LIN{ E6POS: X 728.6422, Y 47.5546, Z -92.0150, A 0, B 90, C 0, E1 0, E2 0, E3 0, E4 0 } C_DIS
LIN{ E6POS: X 729.6150, Y 47.3233, Z -92.0150, A 0, B 90, C 0, E1 0, E2 0, E3 0, E4 0 } C_DIS
LIN{ E6POS: X 730.5879, Y 47.0919, Z -92.0150, A 0, B 90, C 0, E1 0, E2 0, E3 0, E4 0 } C_DIS
LIN{ E6POS: X 731.5608, Y 46.8606, Z -92.0150, A 0, B 90, C 0, E1 0, E2 0, E3 0, E4 0 } C_DIS
LIN{ E6POS: X 731.5744, Y 46.8574, Z -92.0150, A 0, B 90, C 0, E1 0, E2 0, E3 0, E4 0 } C_DIS
LIN{ E6POS: X 732.5446, Y 46.6148, Z -92.0150, A 0, B 90, C 0, E1 0, E2 0, E3 0, E4 0 } C_DIS
LIN{ E6POS: X 733.5147, Y 46.3723, Z -92.0150, A 0, B 90, C 0, E1 0, E2 0, E3 0, E4 0 } C_DIS
LIN{ E6POS: X 734.4849, Y 46.1297, Z -92.0150, A 0, B 90, C 0, E1 0, E2 0, E3 0, E4 0 } C_DIS
LIN{ E6POS: X 735.4550, Y 45.8872, Z -92.0150, A 0, B 90, C 0, E1 0, E2 0, E3 0, E4 0 } C_DIS
LIN{ E6POS: X 736.4251, Y 45.6447, Z -92.0150, A 0, B 90, C 0, E1 0, E2 0, E3 0, E4 0 } C_DIS
LIN{ E6POS: X 737.3953, Y 45.4021, Z -92.0150, A 0, B 90, C 0, E1 0, E2 0, E3 0, E4 0 } C_DIS
LIN{ E6POS: X 738.3654, Y 45.1596, Z -92.0150, A 0, B 90, C 0, E1 0, E2 0, E3 0, E4 0 } C_DIS
LIN{ E6POS: X 739.3356, Y 44.9170, Z -92.0150, A 0, B 90, C 0, E1 0, E2 0, E3 0, E4 0 } C_DIS
LIN{ E6POS: X 740.3057, Y 44.6745, Z -92.0150, A 0, B 90, C 0, E1 0, E2 0, E3 0, E4 0 } C_DIS
LIN{ E6POS: X 740.8582, Y 44.5364, Z -92.0150, A 0, B 90, C 0, E1 0, E2 0, E3 0, E4 0 } C_DIS
LIN{ E6POS: X 741.8351, Y 44.3226, Z -92.0150, A 0, B 90, C 0, E1 0, E2 0, E3 0, E4 0 } C_DIS
LIN{ E6POS: X 742.8120, Y 44.1088, Z -92.0150, A 0, B 90, C 0, E1 0, E2 0, E3 0, E4 0 } C_DIS
LIN{ E6POS: X 743.7889, Y 43.8950, Z -92.0150, A 0, B 90, C 0, E1 0, E2 0, E3 0, E4 0 } C_DIS
LIN{ E6POS: X 744.7658, Y 43.6813, Z -92.0150, A 0, B 90, C 0, E1 0, E2 0, E3 0, E4 0 } C_DIS
LIN{ E6POS: X 744.9749, Y 43.6355, Z -92.0150, A 0, B 90, C 0, E1 0, E2 0, E3 0, E4 0 } C_DIS
LIN{ E6POS: X 745.9497, Y 43.4121, Z -92.0150, A 0, B 90, C 0, E1 0, E2 0, E3 0, E4 0 } C_DIS
LIN{ E6POS: X 746.9244, Y 43.1888, Z -92.0150, A 0, B 90, C 0, E1 0, E2 0, E3 0, E4 0 } C_DIS
LIN{ E6POS: X 747.8991, Y 42.9654, Z -92.0150, A 0, B 90, C 0, E1 0, E2 0, E3 0, E4 0 } C_DIS
LIN{ E6POS: X 748.8739, Y 42.7421, Z -92.0150, A 0, B 90, C 0, E1 0, E2 0, E3 0, E4 0 } C_DIS
LIN{ E6POS: X 749.8486, Y 42.5187, Z -92.0150, A 0, B 90, C 0, E1 0, E2 0, E3 0, E4 0 } C_DIS
LIN{ E6POS: X 750.8233, Y 42.2954, Z -92.0150, A 0, B 90, C 0, E1 0, E2 0, E3 0, E4 0 } C_DIS
LIN{ E6POS: X 751.7981, Y 42.0720, Z -92.0150, A 0, B 90, C 0, E1 0, E2 0, E3 0, E4 0 } C_DIS
LIN{ E6POS: X 752.7728, Y 41.8487, Z -92.0150, A 0, B 90, C 0, E1 0, E2 0, E3 0, E4 0 } C_DIS
LIN{ E6POS: X 753.7476, Y 41.6253, Z -92.0150, A 0, B 90, C 0, E1 0, E2 0, E3 0, E4 0 } C_DIS
LIN{ E6POS: X 754.7223, Y 41.4020, Z -92.0150, A 0, B 90, C 0, E1 0, E2 0, E3 0, E4 0 } C_DIS
LIN{ E6POS: X 754.8028, Y 41.3835, Z -92.0150, A 0, B 90, C 0, E1 0, E2 0, E3 0, E4 0 } C_DIS
LIN{ E6POS: X 755.7861, Y 41.2018, Z -92.0150, A 0, B 90, C 0, E1 0, E2 0, E3 0, E4 0 } C_DIS
LIN{ E6POS: X 756.7695, Y 41.0200, Z -92.0150, A 0, B 90, C 0, E1 0, E2 0, E3 0, E4 0 } C_DIS
LIN{ E6POS: X 757.7528, Y 40.8382, Z -92.0150, A 0, B 90, C 0, E1 0, E2 0, E3 0, E4 0 } C_DIS
LIN{ E6POS: X 758.6031, Y 40.6810, Z -92.0150, A 0, B 90, C 0, E1 0, E2 0, E3 0, E4 0 } C_DIS
LIN{ E6POS: X 759.5852, Y 40.4926, Z -92.0150, A 0, B 90, C 0, E1 0, E2 0, E3 0, E4 0 } C_DIS
LIN{ E6POS: X 760.5673, Y 40.3042, Z -92.0150, A 0, B 90, C 0, E1 0, E2 0, E3 0, E4 0 } C_DIS
LIN{ E6POS: X 761.5493, Y 40.1158, Z -92.0150, A 0, B 90, C 0, E1 0, E2 0, E3 0, E4 0 } C_DIS
LIN{ E6POS: X 762.5314, Y 39.9273, Z -92.0150, A 0, B 90, C 0, E1 0, E2 0, E3 0, E4 0 } C_DIS
LIN{ E6POS: X 763.5135, Y 39.7389, Z -92.0150, A 0, B 90, C 0, E1 0, E2 0, E3 0, E4 0 } C_DIS
LIN{ E6POS: X 764.4956, Y 39.5505, Z -92.0150, A 0, B 90, C 0, E1 0, E2 0, E3 0, E4 0 } C_DIS
LIN{ E6POS: X 765.4777, Y 39.3620, Z -92.0150, A 0, B 90, C 0, E1 0, E2 0, E3 0, E4 0 } C_DIS
LIN{ E6POS: X 766.4598, Y 39.1736, Z -92.0150, A 0, B 90, C 0, E1 0, E2 0, E3 0, E4 0 } C_DIS
LIN{ E6POS: X 767.4419, Y 38.9852, Z -92.0150, A 0, B 90, C 0, E1 0, E2 0, E3 0, E4 0 } C_DIS
LIN{ E6POS: X 767.7439, Y 38.9272, Z -92.0150, A 0, B 90, C 0, E1 0, E2 0, E3 0, E4 0 } C_DIS
LIN{ E6POS: X 768.7376, Y 38.8152, Z -92.0150, A 0, B 90, C 0, E1 0, E2 0, E3 0, E4 0 } C_DIS
LIN{ E6POS: X 769.7313, Y 38.7031, Z -92.0150, A 0, B 90, C 0, E1 0, E2 0, E3 0, E4 0 } C_DIS
LIN{ E6POS: X 770.7009, Y 38.5937, Z -92.0150, A 0, B 90, C 0, E1 0, E2 0, E3 0, E4 0 } C_DIS
LIN{ E6POS: X 771.6945, Y 38.4801, Z -92.0150, A 0, B 90, C 0, E1 0, E2 0, E3 0, E4 0 } C_DIS
LIN{ E6POS: X 772.6880, Y 38.3664, Z -92.0150, A 0, B 90, C 0, E1 0, E2 0, E3 0, E4 0 } C_DIS
LIN{ E6POS: X 773.6815, Y 38.2528, Z -92.0150, A 0, B 90, C 0, E1 0, E2 0, E3 0, E4 0 } C_DIS
LIN{ E6POS: X 774.6750, Y 38.1391, Z -92.0150, A 0, B 90, C 0, E1 0, E2 0, E3 0, E4 0 } C_DIS
LIN{ E6POS: X 775.6686, Y 38.0255, Z -92.0150, A 0, B 90, C 0, E1 0, E2 0, E3 0, E4 0 } C_DIS
LIN{ E6POS: X 776.6621, Y 37.9118, Z -92.0150, A 0, B 90, C 0, E1 0, E2 0, E3 0, E4 0 } C_DIS
LIN{ E6POS: X 777.6556, Y 37.7982, Z -92.0150, A 0, B 90, C 0, E1 0, E2 0, E3 0, E4 0 } C_DIS
LIN{ E6POS: X 777.9256, Y 37.7673, Z -92.0150, A 0, B 90, C 0, E1 0, E2 0, E3 0, E4 0 } C_DIS
LIN{ E6POS: X 778.9253, Y 37.7428, Z -92.0150, A 0, B 90, C 0, E1 0, E2 0, E3 0, E4 0 } C_DIS
LIN{ E6POS: X 779.9250, Y 37.7183, Z -92.0150, A 0, B 90, C 0, E1 0, E2 0, E3 0, E4 0 } C_DIS
LIN{ E6POS: X 780.2499, Y 37.7103, Z -92.0150, A 0, B 90, C 0, E1 0, E2 0, E3 0, E4 0 } C_DIS
LIN{ E6POS: X 781.2496, Y 37.6878, Z -92.0150, A 0, B 90, C 0, E1 0, E2 0, E3 0, E4 0 } C_DIS
LIN{ E6POS: X 782.2494, Y 37.6652, Z -92.0150, A 0, B 90, C 0, E1 0, E2 0, E3 0, E4 0 } C_DIS
LIN{ E6POS: X 783.2491, Y 37.6427, Z -92.0150, A 0, B 90, C 0, E1 0, E2 0, E3 0, E4 0 } C_DIS
LIN{ E6POS: X 784.2489, Y 37.6202, Z -92.0150, A 0, B 90, C 0, E1 0, E2 0, E3 0, E4 0 } C_DIS
LIN{ E6POS: X 785.2486, Y 37.5976, Z -92.0150, A 0, B 90, C 0, E1 0, E2 0, E3 0, E4 0 } C_DIS
LIN{ E6POS: X 786.0367, Y 37.5799, Z -92.0150, A 0, B 90, C 0, E1 0, E2 0, E3 0, E4 0 } C_DIS
LIN{ E6POS: X 787.0345, Y 37.6467, Z -92.0150, A 0, B 90, C 0, E1 0, E2 0, E3 0, E4 0 } C_DIS
LIN{ E6POS: X 787.9393, Y 37.7074, Z -92.0150, A 0, B 90, C 0, E1 0, E2 0, E3 0, E4 0 } C_DIS
LIN{ E6POS: X 788.9369, Y 37.7763, Z -92.0150, A 0, B 90, C 0, E1 0, E2 0, E3 0, E4 0 } C_DIS
LIN{ E6POS: X 789.9345, Y 37.8452, Z -92.0150, A 0, B 90, C 0, E1 0, E2 0, E3 0, E4 0 } C_DIS
LIN{ E6POS: X 790.9321, Y 37.9141, Z -92.0150, A 0, B 90, C 0, E1 0, E2 0, E3 0, E4 0 } C_DIS
LIN{ E6POS: X 791.9298, Y 37.9830, Z -92.0150, A 0, B 90, C 0, E1 0, E2 0, E3 0, E4 0 } C_DIS
LIN{ E6POS: X 792.7685, Y 38.0409, Z -92.0150, A 0, B 90, C 0, E1 0, E2 0, E3 0, E4 0 } C_DIS
LIN{ E6POS: X 793.7601, Y 38.1698, Z -92.0150, A 0, B 90, C 0, E1 0, E2 0, E3 0, E4 0 } C_DIS
LIN{ E6POS: X 794.4600, Y 38.2607, Z -92.0150, A 0, B 90, C 0, E1 0, E2 0, E3 0, E4 0 } C_DIS
LIN{ E6POS: X 795.4517, Y 38.3896, Z -92.0150, A 0, B 90, C 0, E1 0, E2 0, E3 0, E4 0 } C_DIS
LIN{ E6POS: X 796.4433, Y 38.5185, Z -92.0150, A 0, B 90, C 0, E1 0, E2 0, E3 0, E4 0 } C_DIS
LIN{ E6POS: X 797.4350, Y 38.6474, Z -92.0150, A 0, B 90, C 0, E1 0, E2 0, E3 0, E4 0 } C_DIS
LIN{ E6POS: X 798.4266, Y 38.7762, Z -92.0150, A 0, B 90, C 0, E1 0, E2 0, E3 0, E4 0 } C_DIS
LIN{ E6POS: X 798.8097, Y 38.8260, Z -90.0150, A 0, B 90, C 0, E1 0, E2 0, E3 0, E4 0 } C_DIS
LIN{ E6POS: X 798.7068, Y 37.8313, Z -90.0150, A 0, B 90, C 0, E1 0, E2 0, E3 0, E4 0 } C_DIS
LIN{ E6POS: X 798.6040, Y 36.8366, Z -90.0150, A 0, B 90, C 0, E1 0, E2 0, E3 0, E4 0 } C_DIS
LIN{ E6POS: X 798.5012, Y 35.8419, Z -90.0150, A 0, B 90, C 0, E1 0, E2 0, E3 0, E4 0 } C_DIS
LIN{ E6POS: X 798.3983, Y 34.8472, Z -90.0150, A 0, B 90, C 0, E1 0, E2 0, E3 0, E4 0 } C_DIS
LIN{ E6POS: X 798.2955, Y 33.8525, Z -90.0150, A 0, B 90, C 0, E1 0, E2 0, E3 0, E4 0 } C_DIS
LIN{ E6POS: X 798.2022, Y 32.9505, Z -90.0150, A 0, B 90, C 0, E1 0, E2 0, E3 0, E4 0 } C_DIS
LIN{ E6POS: X 798.0994, Y 31.9558, Z -90.0150, A 0, B 90, C 0, E1 0, E2 0, E3 0, E4 0 } C_DIS
LIN{ E6POS: X 797.9966, Y 30.9611, Z -90.0150, A 0, B 90, C 0, E1 0, E2 0, E3 0, E4 0 } C_DIS
LIN{ E6POS: X 797.8938, Y 29.9664, Z -90.0150, A 0, B 90, C 0, E1 0, E2 0, E3 0, E4 0 } C_DIS
LIN{ E6POS: X 797.7909, Y 28.9717, Z -90.0150, A 0, B 90, C 0, E1 0, E2 0, E3 0, E4 0 } C_DIS
LIN{ E6POS: X 797.6881, Y 27.9770, Z -90.0150, A 0, B 90, C 0, E1 0, E2 0, E3 0, E4 0 } C_DIS
LIN{ E6POS: X 797.5853, Y 26.9823, Z -90.0150, A 0, B 90, C 0, E1 0, E2 0, E3 0, E4 0 } C_DIS
LIN{ E6POS: X 797.4824, Y 25.9876, Z -90.0150, A 0, B 90, C 0, E1 0, E2 0, E3 0, E4 0 } C_DIS
LIN{ E6POS: X 797.3796, Y 24.9929, Z -90.0150, A 0, B 90, C 0, E1 0, E2 0, E3 0, E4 0 } C_DIS
LIN{ E6POS: X 797.2768, Y 23.9982, Z -90.0150, A 0, B 90, C 0, E1 0, E2 0, E3 0, E4 0 } C_DIS
LIN{ E6POS: X 797.1739, Y 23.0035, Z -90.0150, A 0, B 90, C 0, E1 0, E2 0, E3 0, E4 0 } C_DIS
LIN{ E6POS: X 797.1224, Y 22.5051, Z -90.0150, A 0, B 90, C 0, E1 0, E2 0, E3 0, E4 0 } C_DIS
LIN{ E6POS: X 797.0002, Y 21.5126, Z -90.0150, A 0, B 90, C 0, E1 0, E2 0, E3 0, E4 0 } C_DIS
LIN{ E6POS: X 796.8780, Y 20.5201, Z -90.0150, A 0, B 90, C 0, E1 0, E2 0, E3 0, E4 0 } C_DIS
LIN{ E6POS: X 796.7559, Y 19.5276, Z -90.0150, A 0, B 90, C 0, E1 0, E2 0, E3 0, E4 0 } C_DIS
LIN{ E6POS: X 796.6337, Y 18.5351, Z -90.0150, A 0, B 90, C 0, E1 0, E2 0, E3 0, E4 0 } C_DIS
LIN{ E6POS: X 796.5115, Y 17.5426, Z -90.0150, A 0, B 90, C 0, E1 0, E2 0, E3 0, E4 0 } C_DIS
LIN{ E6POS: X 796.4506, Y 17.0475, Z -90.0150, A 0, B 90, C 0, E1 0, E2 0, E3 0, E4 0 } C_DIS
LIN{ E6POS: X 796.3284, Y 16.0550, Z -90.0150, A 0, B 90, C 0, E1 0, E2 0, E3 0, E4 0 } C_DIS
LIN{ E6POS: X 796.2062, Y 15.0625, Z -90.0150, A 0, B 90, C 0, E1 0, E2 0, E3 0, E4 0 } C_DIS
LIN{ E6POS: X 796.0840, Y 14.0700, Z -90.0150, A 0, B 90, C 0, E1 0, E2 0, E3 0, E4 0 } C_DIS
LIN{ E6POS: X 795.9619, Y 13.0775, Z -90.0150, A 0, B 90, C 0, E1 0, E2 0, E3 0, E4 0 } C_DIS
LIN{ E6POS: X 795.8397, Y 12.0850, Z -90.0150, A 0, B 90, C 0, E1 0, E2 0, E3 0, E4 0 } C_DIS
LIN{ E6POS: X 795.7175, Y 11.0925, Z -90.0150, A 0, B 90, C 0, E1 0, E2 0, E3 0, E4 0 } C_DIS
LIN{ E6POS: X 795.5953, Y 10.1000, Z -90.0150, A 0, B 90, C 0, E1 0, E2 0, E3 0, E4 0 } C_DIS
LIN{ E6POS: X 795.4732, Y 9.1075, Z -90.0150, A 0, B 90, C 0, E1 0, E2 0, E3 0, E4 0 } C_DIS
LIN{ E6POS: X 795.3510, Y 8.1150, Z -90.0150, A 0, B 90, C 0, E1 0, E2 0, E3 0, E4 0 } C_DIS
LIN{ E6POS: X 795.2562, Y 7.3452, Z -90.0150, A 0, B 90, C 0, E1 0, E2 0, E3 0, E4 0 } C_DIS
LIN{ E6POS: X 795.0854, Y 6.3599, Z -90.0150, A 0, B 90, C 0, E1 0, E2 0, E3 0, E4 0 } C_DIS
LIN{ E6POS: X 794.9146, Y 5.3746, Z -90.0150, A 0, B 90, C 0, E1 0, E2 0, E3 0, E4 0 } C_DIS
LIN{ E6POS: X 794.7438, Y 4.3893, Z -90.0150, A 0, B 90, C 0, E1 0, E2 0, E3 0, E4 0 } C_DIS
LIN{ E6POS: X 794.5730, Y 3.4040, Z -90.0150, A 0, B 90, C 0, E1 0, E2 0, E3 0, E4 0 } C_DIS
LIN{ E6POS: X 794.4552, Y 2.7245, Z -90.0150, A 0, B 90, C 0, E1 0, E2 0, E3 0, E4 0 } C_DIS
LIN{ E6POS: X 794.2843, Y 1.7392, Z -90.0150, A 0, B 90, C 0, E1 0, E2 0, E3 0, E4 0 } C_DIS
LIN{ E6POS: X 794.1135, Y 0.7539, Z -90.0150, A 0, B 90, C 0, E1 0, E2 0, E3 0, E4 0 } C_DIS
LIN{ E6POS: X 793.9427, Y -0.2314, Z -90.0150, A 0, B 90, C 0, E1 0, E2 0, E3 0, E4 0 } C_DIS
LIN{ E6POS: X 793.7719, Y -1.2167, Z -90.0150, A 0, B 90, C 0, E1 0, E2 0, E3 0, E4 0 } C_DIS
LIN{ E6POS: X 793.6011, Y -2.2020, Z -90.0150, A 0, B 90, C 0, E1 0, E2 0, E3 0, E4 0 } C_DIS
LIN{ E6POS: X 793.4303, Y -3.1873, Z -90.0150, A 0, B 90, C 0, E1 0, E2 0, E3 0, E4 0 } C_DIS
LIN{ E6POS: X 793.2594, Y -4.1726, Z -90.0150, A 0, B 90, C 0, E1 0, E2 0, E3 0, E4 0 } C_DIS
LIN{ E6POS: X 793.0886, Y -5.1579, Z -90.0150, A 0, B 90, C 0, E1 0, E2 0, E3 0, E4 0 } C_DIS
LIN{ E6POS: X 793.0310, Y -5.4900, Z -90.0150, A 0, B 90, C 0, E1 0, E2 0, E3 0, E4 0 } C_DIS
LIN{ E6POS: X 792.7476, Y -6.4490, Z -90.0150, A 0, B 90, C 0, E1 0, E2 0, E3 0, E4 0 } C_DIS
LIN{ E6POS: X 792.4642, Y -7.4080, Z -90.0150, A 0, B 90, C 0, E1 0, E2 0, E3 0, E4 0 } C_DIS
LIN{ E6POS: X 792.1808, Y -8.3670, Z -90.0150, A 0, B 90, C 0, E1 0, E2 0, E3 0, E4 0 } C_DIS
LIN{ E6POS: X 792.0364, Y -8.8556, Z -90.0150, A 0, B 90, C 0, E1 0, E2 0, E3 0, E4 0 } C_DIS
LIN{ E6POS: X 791.7530, Y -9.8146, Z -90.0150, A 0, B 90, C 0, E1 0, E2 0, E3 0, E4 0 } C_DIS
LIN{ E6POS: X 791.4696, Y -10.7736, Z -90.0150, A 0, B 90, C 0, E1 0, E2 0, E3 0, E4 0 } C_DIS
LIN{ E6POS: X 791.1861, Y -11.7326, Z -90.0150, A 0, B 90, C 0, E1 0, E2 0, E3 0, E4 0 } C_DIS
LIN{ E6POS: X 790.9027, Y -12.6916, Z -90.0150, A 0, B 90, C 0, E1 0, E2 0, E3 0, E4 0 } C_DIS
LIN{ E6POS: X 790.6193, Y -13.6506, Z -90.0150, A 0, B 90, C 0, E1 0, E2 0, E3 0, E4 0 } C_DIS
LIN{ E6POS: X 790.3359, Y -14.6096, Z -90.0150, A 0, B 90, C 0, E1 0, E2 0, E3 0, E4 0 } C_DIS
LIN{ E6POS: X 790.2681, Y -14.8387, Z -90.0150, A 0, B 90, C 0, E1 0, E2 0, E3 0, E4 0 } C_DIS
LIN{ E6POS: X 789.6733, Y -15.6426, Z -90.0150, A 0, B 90, C 0, E1 0, E2 0, E3 0, E4 0 } C_DIS
LIN{ E6POS: X 789.0784, Y -16.4464, Z -90.0150, A 0, B 90, C 0, E1 0, E2 0, E3 0, E4 0 } C_DIS
LIN{ E6POS: X 789.0154, Y -16.5315, Z -90.0150, A 0, B 90, C 0, E1 0, E2 0, E3 0, E4 0 } C_DIS
LIN{ E6POS: X 788.4206, Y -17.3353, Z -90.0150, A 0, B 90, C 0, E1 0, E2 0, E3 0, E4 0 } C_DIS
LIN{ E6POS: X 787.8257, Y -18.1391, Z -90.0150, A 0, B 90, C 0, E1 0, E2 0, E3 0, E4 0 } C_DIS
LIN{ E6POS: X 787.2308, Y -18.9429, Z -90.0150, A 0, B 90, C 0, E1 0, E2 0, E3 0, E4 0 } C_DIS
LIN{ E6POS: X 786.7884, Y -19.5408, Z -90.0150, A 0, B 90, C 0, E1 0, E2 0, E3 0, E4 0 } C_DIS
LIN{ E6POS: X 785.8300, Y -19.8262, Z -90.0150, A 0, B 90, C 0, E1 0, E2 0, E3 0, E4 0 } C_DIS
LIN{ E6POS: X 785.1744, Y -20.0215, Z -90.0150, A 0, B 90, C 0, E1 0, E2 0, E3 0, E4 0 } C_DIS
LIN{ E6POS: X 784.2171, Y -20.3108, Z -90.0150, A 0, B 90, C 0, E1 0, E2 0, E3 0, E4 0 } C_DIS
LIN{ E6POS: X 783.2598, Y -20.6000, Z -90.0150, A 0, B 90, C 0, E1 0, E2 0, E3 0, E4 0 } C_DIS
LIN{ E6POS: X 782.3421, Y -20.8773, Z -90.0150, A 0, B 90, C 0, E1 0, E2 0, E3 0, E4 0 } C_DIS
LIN{ E6POS: X 781.3508, Y -20.7456, Z -90.0150, A 0, B 90, C 0, E1 0, E2 0, E3 0, E4 0 } C_DIS
LIN{ E6POS: X 780.3595, Y -20.6140, Z -90.0150, A 0, B 90, C 0, E1 0, E2 0, E3 0, E4 0 } C_DIS
LIN{ E6POS: X 779.3682, Y -20.4824, Z -90.0150, A 0, B 90, C 0, E1 0, E2 0, E3 0, E4 0 } C_DIS
LIN{ E6POS: X 778.7599, Y -20.4017, Z -90.0150, A 0, B 90, C 0, E1 0, E2 0, E3 0, E4 0 } C_DIS
LIN{ E6POS: X 777.7682, Y -20.2731, Z -90.0150, A 0, B 90, C 0, E1 0, E2 0, E3 0, E4 0 } C_DIS
LIN{ E6POS: X 776.7765, Y -20.1446, Z -90.0150, A 0, B 90, C 0, E1 0, E2 0, E3 0, E4 0 } C_DIS
LIN{ E6POS: X 776.6816, Y -20.1323, Z -90.0150, A 0, B 90, C 0, E1 0, E2 0, E3 0, E4 0 } C_DIS
LIN{ E6POS: X 775.7050, Y -19.9174, Z -90.0150, A 0, B 90, C 0, E1 0, E2 0, E3 0, E4 0 } C_DIS
LIN{ E6POS: X 774.7283, Y -19.7025, Z -90.0150, A 0, B 90, C 0, E1 0, E2 0, E3 0, E4 0 } C_DIS
LIN{ E6POS: X 773.7517, Y -19.4876, Z -90.0150, A 0, B 90, C 0, E1 0, E2 0, E3 0, E4 0 } C_DIS
LIN{ E6POS: X 772.7751, Y -19.2728, Z -90.0150, A 0, B 90, C 0, E1 0, E2 0, E3 0, E4 0 } C_DIS
LIN{ E6POS: X 772.2027, Y -19.1468, Z -90.0150, A 0, B 90, C 0, E1 0, E2 0, E3 0, E4 0 } C_DIS
LIN{ E6POS: X 771.2243, Y -18.9404, Z -90.0150, A 0, B 90, C 0, E1 0, E2 0, E3 0, E4 0 } C_DIS
LIN{ E6POS: X 770.2458, Y -18.7339, Z -90.0150, A 0, B 90, C 0, E1 0, E2 0, E3 0, E4 0 } C_DIS
LIN{ E6POS: X 769.5569, Y -18.5885, Z -90.0150, A 0, B 90, C 0, E1 0, E2 0, E3 0, E4 0 } C_DIS
LIN{ E6POS: X 768.5642, Y -18.4673, Z -90.0150, A 0, B 90, C 0, E1 0, E2 0, E3 0, E4 0 } C_DIS
LIN{ E6POS: X 767.5716, Y -18.3462, Z -90.0150, A 0, B 90, C 0, E1 0, E2 0, E3 0, E4 0 } C_DIS
LIN{ E6POS: X 766.5790, Y -18.2251, Z -90.0150, A 0, B 90, C 0, E1 0, E2 0, E3 0, E4 0 } C_DIS
LIN{ E6POS: X 765.5863, Y -18.1039, Z -90.0150, A 0, B 90, C 0, E1 0, E2 0, E3 0, E4 0 } C_DIS
LIN{ E6POS: X 764.5937, Y -17.9828, Z -90.0150, A 0, B 90, C 0, E1 0, E2 0, E3 0, E4 0 } C_DIS
LIN{ E6POS: X 764.0362, Y -17.9147, Z -90.0150, A 0, B 90, C 0, E1 0, E2 0, E3 0, E4 0 } C_DIS
LIN{ E6POS: X 763.0429, Y -17.7993, Z -90.0150, A 0, B 90, C 0, E1 0, E2 0, E3 0, E4 0 } C_DIS
LIN{ E6POS: X 762.0496, Y -17.6838, Z -90.0150, A 0, B 90, C 0, E1 0, E2 0, E3 0, E4 0 } C_DIS
LIN{ E6POS: X 761.0563, Y -17.5683, Z -90.0150, A 0, B 90, C 0, E1 0, E2 0, E3 0, E4 0 } C_DIS
LIN{ E6POS: X 760.7202, Y -17.5293, Z -90.0150, A 0, B 90, C 0, E1 0, E2 0, E3 0, E4 0 } C_DIS
LIN{ E6POS: X 759.7223, Y -17.4645, Z -90.0150, A 0, B 90, C 0, E1 0, E2 0, E3 0, E4 0 } C_DIS
LIN{ E6POS: X 758.7244, Y -17.3998, Z -90.0150, A 0, B 90, C 0, E1 0, E2 0, E3 0, E4 0 } C_DIS
LIN{ E6POS: X 757.7265, Y -17.3350, Z -90.0150, A 0, B 90, C 0, E1 0, E2 0, E3 0, E4 0 } C_DIS
LIN{ E6POS: X 756.7286, Y -17.2703, Z -90.0150, A 0, B 90, C 0, E1 0, E2 0, E3 0, E4 0 } C_DIS
LIN{ E6POS: X 755.7307, Y -17.2056, Z -90.0150, A 0, B 90, C 0, E1 0, E2 0, E3 0, E4 0 } C_DIS
LIN{ E6POS: X 754.8606, Y -17.1491, Z -90.0150, A 0, B 90, C 0, E1 0, E2 0, E3 0, E4 0 } C_DIS
LIN{ E6POS: X 753.8626, Y -17.0864, Z -90.0150, A 0, B 90, C 0, E1 0, E2 0, E3 0, E4 0 } C_DIS
LIN{ E6POS: X 752.8645, Y -17.0237, Z -90.0150, A 0, B 90, C 0, E1 0, E2 0, E3 0, E4 0 } C_DIS
LIN{ E6POS: X 751.8665, Y -16.9611, Z -90.0150, A 0, B 90, C 0, E1 0, E2 0, E3 0, E4 0 } C_DIS
LIN{ E6POS: X 751.3122, Y -16.9262, Z -90.0150, A 0, B 90, C 0, E1 0, E2 0, E3 0, E4 0 } C_DIS
LIN{ E6POS: X 750.3124, Y -16.9073, Z -90.0150, A 0, B 90, C 0, E1 0, E2 0, E3 0, E4 0 } C_DIS
LIN{ E6POS: X 749.3126, Y -16.8884, Z -90.0150, A 0, B 90, C 0, E1 0, E2 0, E3 0, E4 0 } C_DIS
LIN{ E6POS: X 748.3128, Y -16.8695, Z -90.0150, A 0, B 90, C 0, E1 0, E2 0, E3 0, E4 0 } C_DIS
LIN{ E6POS: X 747.3130, Y -16.8506, Z -90.0150, A 0, B 90, C 0, E1 0, E2 0, E3 0, E4 0 } C_DIS
LIN{ E6POS: X 746.3131, Y -16.8317, Z -90.0150, A 0, B 90, C 0, E1 0, E2 0, E3 0, E4 0 } C_DIS
LIN{ E6POS: X 745.8162, Y -16.8224, Z -90.0150, A 0, B 90, C 0, E1 0, E2 0, E3 0, E4 0 } C_DIS
LIN{ E6POS: X 744.8164, Y -16.8011, Z -90.0150, A 0, B 90, C 0, E1 0, E2 0, E3 0, E4 0 } C_DIS
LIN{ E6POS: X 743.8167, Y -16.7799, Z -90.0150, A 0, B 90, C 0, E1 0, E2 0, E3 0, E4 0 } C_DIS
LIN{ E6POS: X 742.8169, Y -16.7587, Z -90.0150, A 0, B 90, C 0, E1 0, E2 0, E3 0, E4 0 } C_DIS
LIN{ E6POS: X 742.4732, Y -16.7514, Z -90.0150, A 0, B 90, C 0, E1 0, E2 0, E3 0, E4 0 } C_DIS
LIN{ E6POS: X 741.4738, Y -16.7860, Z -90.0150, A 0, B 90, C 0, E1 0, E2 0, E3 0, E4 0 } C_DIS
LIN{ E6POS: X 740.4744, Y -16.8206, Z -90.0150, A 0, B 90, C 0, E1 0, E2 0, E3 0, E4 0 } C_DIS
LIN{ E6POS: X 739.4750, Y -16.8552, Z -90.0150, A 0, B 90, C 0, E1 0, E2 0, E3 0, E4 0 } C_DIS
LIN{ E6POS: X 738.4756, Y -16.8898, Z -90.0150, A 0, B 90, C 0, E1 0, E2 0, E3 0, E4 0 } C_DIS
LIN{ E6POS: X 738.0444, Y -16.9047, Z -90.0150, A 0, B 90, C 0, E1 0, E2 0, E3 0, E4 0 } C_DIS
LIN{ E6POS: X 737.0448, Y -16.9308, Z -90.0150, A 0, B 90, C 0, E1 0, E2 0, E3 0, E4 0 } C_DIS
LIN{ E6POS: X 736.0451, Y -16.9570, Z -90.0150, A 0, B 90, C 0, E1 0, E2 0, E3 0, E4 0 } C_DIS
LIN{ E6POS: X 735.3446, Y -16.9753, Z -90.0150, A 0, B 90, C 0, E1 0, E2 0, E3 0, E4 0 } C_DIS
LIN{ E6POS: X 734.3554, Y -17.1219, Z -90.0150, A 0, B 90, C 0, E1 0, E2 0, E3 0, E4 0 } C_DIS
LIN{ E6POS: X 733.3662, Y -17.2684, Z -90.0150, A 0, B 90, C 0, E1 0, E2 0, E3 0, E4 0 } C_DIS
LIN{ E6POS: X 732.6860, Y -17.3692, Z -90.0150, A 0, B 90, C 0, E1 0, E2 0, E3 0, E4 0 } C_DIS
LIN{ E6POS: X 731.6937, Y -17.4931, Z -90.0150, A 0, B 90, C 0, E1 0, E2 0, E3 0, E4 0 } C_DIS
LIN{ E6POS: X 731.0673, Y -17.5712, Z -90.0150, A 0, B 90, C 0, E1 0, E2 0, E3 0, E4 0 } C_DIS
LIN{ E6POS: X 730.2510, Y -18.1489, Z -90.0150, A 0, B 90, C 0, E1 0, E2 0, E3 0, E4 0 } C_DIS
LIN{ E6POS: X 730.1785, Y -18.2002, Z -90.0150, A 0, B 90, C 0, E1 0, E2 0, E3 0, E4 0 } C_DIS
LIN{ E6POS: X 729.6399, Y -18.5352, Z -90.0150, A 0, B 90, C 0, E1 0, E2 0, E3 0, E4 0 } C_DIS
LIN{ E6POS: X 730.1801, Y -19.0046, Z -90.0150, A 0, B 90, C 0, E1 0, E2 0, E3 0, E4 0 } C_DIS
LIN{ E6POS: X 730.8967, Y -19.7021, Z -90.0150, A 0, B 90, C 0, E1 0, E2 0, E3 0, E4 0 } C_DIS
LIN{ E6POS: X 731.0609, Y -19.8620, Z -90.0150, A 0, B 90, C 0, E1 0, E2 0, E3 0, E4 0 } C_DIS
LIN{ E6POS: X 731.9974, Y -20.2128, Z -90.0150, A 0, B 90, C 0, E1 0, E2 0, E3 0, E4 0 } C_DIS
LIN{ E6POS: X 732.6792, Y -20.4682, Z -90.0150, A 0, B 90, C 0, E1 0, E2 0, E3 0, E4 0 } C_DIS
LIN{ E6POS: X 733.6051, Y -20.8461, Z -90.0150, A 0, B 90, C 0, E1 0, E2 0, E3 0, E4 0 } C_DIS
LIN{ E6POS: X 734.5309, Y -21.2240, Z -90.0150, A 0, B 90, C 0, E1 0, E2 0, E3 0, E4 0 } C_DIS
LIN{ E6POS: X 735.3296, Y -21.5500, Z -90.0150, A 0, B 90, C 0, E1 0, E2 0, E3 0, E4 0 } C_DIS
LIN{ E6POS: X 736.2935, Y -21.8161, Z -90.0150, A 0, B 90, C 0, E1 0, E2 0, E3 0, E4 0 } C_DIS
LIN{ E6POS: X 737.2575, Y -22.0822, Z -90.0150, A 0, B 90, C 0, E1 0, E2 0, E3 0, E4 0 } C_DIS
LIN{ E6POS: X 738.0246, Y -22.2940, Z -90.0150, A 0, B 90, C 0, E1 0, E2 0, E3 0, E4 0 } C_DIS
LIN{ E6POS: X 738.9840, Y -22.5764, Z -90.0150, A 0, B 90, C 0, E1 0, E2 0, E3 0, E4 0 } C_DIS
LIN{ E6POS: X 739.9433, Y -22.8587, Z -90.0150, A 0, B 90, C 0, E1 0, E2 0, E3 0, E4 0 } C_DIS
LIN{ E6POS: X 740.9026, Y -23.1411, Z -90.0150, A 0, B 90, C 0, E1 0, E2 0, E3 0, E4 0 } C_DIS
LIN{ E6POS: X 741.8619, Y -23.4234, Z -90.0150, A 0, B 90, C 0, E1 0, E2 0, E3 0, E4 0 } C_DIS
LIN{ E6POS: X 742.4436, Y -23.5946, Z -90.0150, A 0, B 90, C 0, E1 0, E2 0, E3 0, E4 0 } C_DIS
LIN{ E6POS: X 743.4184, Y -23.8176, Z -90.0150, A 0, B 90, C 0, E1 0, E2 0, E3 0, E4 0 } C_DIS
LIN{ E6POS: X 744.3932, Y -24.0406, Z -90.0150, A 0, B 90, C 0, E1 0, E2 0, E3 0, E4 0 } C_DIS
LIN{ E6POS: X 745.3681, Y -24.2635, Z -90.0150, A 0, B 90, C 0, E1 0, E2 0, E3 0, E4 0 } C_DIS
LIN{ E6POS: X 745.7801, Y -24.3578, Z -90.0150, A 0, B 90, C 0, E1 0, E2 0, E3 0, E4 0 } C_DIS
LIN{ E6POS: X 746.7524, Y -24.5912, Z -90.0150, A 0, B 90, C 0, E1 0, E2 0, E3 0, E4 0 } C_DIS
LIN{ E6POS: X 747.7248, Y -24.8246, Z -90.0150, A 0, B 90, C 0, E1 0, E2 0, E3 0, E4 0 } C_DIS
LIN{ E6POS: X 748.6972, Y -25.0580, Z -90.0150, A 0, B 90, C 0, E1 0, E2 0, E3 0, E4 0 } C_DIS
LIN{ E6POS: X 749.6696, Y -25.2915, Z -90.0150, A 0, B 90, C 0, E1 0, E2 0, E3 0, E4 0 } C_DIS
LIN{ E6POS: X 750.6419, Y -25.5249, Z -90.0150, A 0, B 90, C 0, E1 0, E2 0, E3 0, E4 0 } C_DIS
LIN{ E6POS: X 751.2672, Y -25.6750, Z -90.0150, A 0, B 90, C 0, E1 0, E2 0, E3 0, E4 0 } C_DIS
LIN{ E6POS: X 752.2502, Y -25.8587, Z -90.0150, A 0, B 90, C 0, E1 0, E2 0, E3 0, E4 0 } C_DIS
LIN{ E6POS: X 753.2332, Y -26.0425, Z -90.0150, A 0, B 90, C 0, E1 0, E2 0, E3 0, E4 0 } C_DIS
LIN{ E6POS: X 754.2161, Y -26.2262, Z -90.0150, A 0, B 90, C 0, E1 0, E2 0, E3 0, E4 0 } C_DIS
LIN{ E6POS: X 754.8091, Y -26.3371, Z -90.0150, A 0, B 90, C 0, E1 0, E2 0, E3 0, E4 0 } C_DIS
LIN{ E6POS: X 755.7909, Y -26.5271, Z -90.0150, A 0, B 90, C 0, E1 0, E2 0, E3 0, E4 0 } C_DIS
LIN{ E6POS: X 756.7727, Y -26.7170, Z -90.0150, A 0, B 90, C 0, E1 0, E2 0, E3 0, E4 0 } C_DIS
LIN{ E6POS: X 757.7544, Y -26.9070, Z -90.0150, A 0, B 90, C 0, E1 0, E2 0, E3 0, E4 0 } C_DIS
LIN{ E6POS: X 758.7362, Y -27.0970, Z -90.0150, A 0, B 90, C 0, E1 0, E2 0, E3 0, E4 0 } C_DIS
LIN{ E6POS: X 759.7180, Y -27.2870, Z -90.0150, A 0, B 90, C 0, E1 0, E2 0, E3 0, E4 0 } C_DIS
LIN{ E6POS: X 760.6632, Y -27.4699, Z -90.0150, A 0, B 90, C 0, E1 0, E2 0, E3 0, E4 0 } C_DIS
LIN{ E6POS: X 761.6544, Y -27.6022, Z -90.0150, A 0, B 90, C 0, E1 0, E2 0, E3 0, E4 0 } C_DIS
LIN{ E6POS: X 762.6456, Y -27.7346, Z -90.0150, A 0, B 90, C 0, E1 0, E2 0, E3 0, E4 0 } C_DIS
LIN{ E6POS: X 763.6368, Y -27.8669, Z -90.0150, A 0, B 90, C 0, E1 0, E2 0, E3 0, E4 0 } C_DIS
LIN{ E6POS: X 763.9751, Y -27.9121, Z -90.0150, A 0, B 90, C 0, E1 0, E2 0, E3 0, E4 0 } C_DIS
LIN{ E6POS: X 764.9660, Y -28.0461, Z -90.0150, A 0, B 90, C 0, E1 0, E2 0, E3 0, E4 0 } C_DIS
LIN{ E6POS: X 765.9570, Y -28.1801, Z -90.0150, A 0, B 90, C 0, E1 0, E2 0, E3 0, E4 0 } C_DIS
LIN{ E6POS: X 766.9480, Y -28.3142, Z -90.0150, A 0, B 90, C 0, E1 0, E2 0, E3 0, E4 0 } C_DIS
LIN{ E6POS: X 767.9390, Y -28.4482, Z -90.0150, A 0, B 90, C 0, E1 0, E2 0, E3 0, E4 0 } C_DIS
LIN{ E6POS: X 768.9300, Y -28.5822, Z -90.0150, A 0, B 90, C 0, E1 0, E2 0, E3 0, E4 0 } C_DIS
LIN{ E6POS: X 769.4939, Y -28.6585, Z -90.0150, A 0, B 90, C 0, E1 0, E2 0, E3 0, E4 0 } C_DIS
LIN{ E6POS: X 770.4932, Y -28.6971, Z -90.0150, A 0, B 90, C 0, E1 0, E2 0, E3 0, E4 0 } C_DIS
LIN{ E6POS: X 771.4924, Y -28.7358, Z -90.0150, A 0, B 90, C 0, E1 0, E2 0, E3 0, E4 0 } C_DIS
LIN{ E6POS: X 772.1404, Y -28.7609, Z -90.0150, A 0, B 90, C 0, E1 0, E2 0, E3 0, E4 0 } C_DIS
LIN{ E6POS: X 773.1398, Y -28.7964, Z -90.0150, A 0, B 90, C 0, E1 0, E2 0, E3 0, E4 0 } C_DIS
LIN{ E6POS: X 774.1391, Y -28.8319, Z -90.0150, A 0, B 90, C 0, E1 0, E2 0, E3 0, E4 0 } C_DIS
LIN{ E6POS: X 775.1385, Y -28.8674, Z -90.0150, A 0, B 90, C 0, E1 0, E2 0, E3 0, E4 0 } C_DIS
LIN{ E6POS: X 776.1379, Y -28.9030, Z -90.0150, A 0, B 90, C 0, E1 0, E2 0, E3 0, E4 0 } C_DIS
LIN{ E6POS: X 776.6244, Y -28.9203, Z -90.0150, A 0, B 90, C 0, E1 0, E2 0, E3 0, E4 0 } C_DIS
LIN{ E6POS: X 777.6080, Y -29.1010, Z -90.0150, A 0, B 90, C 0, E1 0, E2 0, E3 0, E4 0 } C_DIS
LIN{ E6POS: X 778.5601, Y -29.2760, Z -90.0150, A 0, B 90, C 0, E1 0, E2 0, E3 0, E4 0 } C_DIS
LIN{ E6POS: X 779.5432, Y -29.4588, Z -90.0150, A 0, B 90, C 0, E1 0, E2 0, E3 0, E4 0 } C_DIS
LIN{ E6POS: X 780.5264, Y -29.6417, Z -90.0150, A 0, B 90, C 0, E1 0, E2 0, E3 0, E4 0 } C_DIS
LIN{ E6POS: X 781.5095, Y -29.8246, Z -90.0150, A 0, B 90, C 0, E1 0, E2 0, E3 0, E4 0 } C_DIS
LIN{ E6POS: X 781.8901, Y -29.8954, Z -90.0150, A 0, B 90, C 0, E1 0, E2 0, E3 0, E4 0 } C_DIS
LIN{ E6POS: X 782.5907, Y -30.6089, Z -90.0150, A 0, B 90, C 0, E1 0, E2 0, E3 0, E4 0 } C_DIS
LIN{ E6POS: X 783.0689, Y -31.0959, Z -90.0150, A 0, B 90, C 0, E1 0, E2 0, E3 0, E4 0 } C_DIS
LIN{ E6POS: X 783.7638, Y -31.8150, Z -90.0150, A 0, B 90, C 0, E1 0, E2 0, E3 0, E4 0 } C_DIS
LIN{ E6POS: X 784.4588, Y -32.5340, Z -90.0150, A 0, B 90, C 0, E1 0, E2 0, E3 0, E4 0 } C_DIS
LIN{ E6POS: X 785.1281, Y -33.2266, Z -90.0150, A 0, B 90, C 0, E1 0, E2 0, E3 0, E4 0 } C_DIS
LIN{ E6POS: X 785.2695, Y -34.2166, Z -90.0150, A 0, B 90, C 0, E1 0, E2 0, E3 0, E4 0 } C_DIS
LIN{ E6POS: X 785.4109, Y -35.2065, Z -90.0150, A 0, B 90, C 0, E1 0, E2 0, E3 0, E4 0 } C_DIS
LIN{ E6POS: X 785.5049, Y -35.8643, Z -90.0150, A 0, B 90, C 0, E1 0, E2 0, E3 0, E4 0 } C_DIS
LIN{ E6POS: X 785.6463, Y -36.8543, Z -90.0150, A 0, B 90, C 0, E1 0, E2 0, E3 0, E4 0 } C_DIS
LIN{ E6POS: X 785.7877, Y -37.8442, Z -90.0150, A 0, B 90, C 0, E1 0, E2 0, E3 0, E4 0 } C_DIS
LIN{ E6POS: X 785.9291, Y -38.8342, Z -90.0150, A 0, B 90, C 0, E1 0, E2 0, E3 0, E4 0 } C_DIS
LIN{ E6POS: X 786.0705, Y -39.8241, Z -90.0150, A 0, B 90, C 0, E1 0, E2 0, E3 0, E4 0 } C_DIS
LIN{ E6POS: X 786.1747, Y -40.5536, Z -90.0150, A 0, B 90, C 0, E1 0, E2 0, E3 0, E4 0 } C_DIS
LIN{ E6POS: X 786.0743, Y -41.5485, Z -90.0150, A 0, B 90, C 0, E1 0, E2 0, E3 0, E4 0 } C_DIS
LIN{ E6POS: X 785.9740, Y -42.5435, Z -90.0150, A 0, B 90, C 0, E1 0, E2 0, E3 0, E4 0 } C_DIS
LIN{ E6POS: X 785.8737, Y -43.5384, Z -90.0150, A 0, B 90, C 0, E1 0, E2 0, E3 0, E4 0 } C_DIS
LIN{ E6POS: X 785.7734, Y -44.5334, Z -90.0150, A 0, B 90, C 0, E1 0, E2 0, E3 0, E4 0 } C_DIS
LIN{ E6POS: X 785.7041, Y -45.2209, Z -90.0150, A 0, B 90, C 0, E1 0, E2 0, E3 0, E4 0 } C_DIS
LIN{ E6POS: X 785.6038, Y -46.2159, Z -90.0150, A 0, B 90, C 0, E1 0, E2 0, E3 0, E4 0 } C_DIS
LIN{ E6POS: X 785.5035, Y -47.2108, Z -90.0150, A 0, B 90, C 0, E1 0, E2 0, E3 0, E4 0 } C_DIS
LIN{ E6POS: X 785.4031, Y -48.2058, Z -90.0150, A 0, B 90, C 0, E1 0, E2 0, E3 0, E4 0 } C_DIS
LIN{ E6POS: X 785.3028, Y -49.2007, Z -90.0150, A 0, B 90, C 0, E1 0, E2 0, E3 0, E4 0 } C_DIS
LIN{ E6POS: X 785.2025, Y -50.1957, Z -90.0150, A 0, B 90, C 0, E1 0, E2 0, E3 0, E4 0 } C_DIS
LIN{ E6POS: X 785.1022, Y -51.1907, Z -90.0150, A 0, B 90, C 0, E1 0, E2 0, E3 0, E4 0 } C_DIS
LIN{ E6POS: X 785.0019, Y -52.1856, Z -90.0150, A 0, B 90, C 0, E1 0, E2 0, E3 0, E4 0 } C_DIS
LIN{ E6POS: X 784.9016, Y -53.1806, Z -90.0150, A 0, B 90, C 0, E1 0, E2 0, E3 0, E4 0 } C_DIS
LIN{ E6POS: X 784.8675, Y -53.5185, Z -90.0150, A 0, B 90, C 0, E1 0, E2 0, E3 0, E4 0 } C_DIS
LIN{ E6POS: X 784.6915, Y -54.5029, Z -90.0150, A 0, B 90, C 0, E1 0, E2 0, E3 0, E4 0 } C_DIS
LIN{ E6POS: X 784.5156, Y -55.4873, Z -90.0150, A 0, B 90, C 0, E1 0, E2 0, E3 0, E4 0 } C_DIS
LIN{ E6POS: X 784.3396, Y -56.4717, Z -90.0150, A 0, B 90, C 0, E1 0, E2 0, E3 0, E4 0 } C_DIS
LIN{ E6POS: X 784.1637, Y -57.4560, Z -90.0150, A 0, B 90, C 0, E1 0, E2 0, E3 0, E4 0 } C_DIS
LIN{ E6POS: X 783.9877, Y -58.4404, Z -90.0150, A 0, B 90, C 0, E1 0, E2 0, E3 0, E4 0 } C_DIS
LIN{ E6POS: X 783.8118, Y -59.4248, Z -90.0150, A 0, B 90, C 0, E1 0, E2 0, E3 0, E4 0 } C_DIS
LIN{ E6POS: X 783.7612, Y -59.7081, Z -90.0150, A 0, B 90, C 0, E1 0, E2 0, E3 0, E4 0 } C_DIS
LIN{ E6POS: X 783.5852, Y -60.6925, Z -90.0150, A 0, B 90, C 0, E1 0, E2 0, E3 0, E4 0 } C_DIS
LIN{ E6POS: X 783.4093, Y -61.6769, Z -90.0150, A 0, B 90, C 0, E1 0, E2 0, E3 0, E4 0 } C_DIS
LIN{ E6POS: X 783.2333, Y -62.6613, Z -90.0150, A 0, B 90, C 0, E1 0, E2 0, E3 0, E4 0 } C_DIS
LIN{ E6POS: X 783.0574, Y -63.6457, Z -90.0150, A 0, B 90, C 0, E1 0, E2 0, E3 0, E4 0 } C_DIS
LIN{ E6POS: X 782.8814, Y -64.6301, Z -90.0150, A 0, B 90, C 0, E1 0, E2 0, E3 0, E4 0 } C_DIS
LIN{ E6POS: X 782.7055, Y -65.6145, Z -90.0150, A 0, B 90, C 0, E1 0, E2 0, E3 0, E4 0 } C_DIS
LIN{ E6POS: X 782.5295, Y -66.5989, Z -90.0150, A 0, B 90, C 0, E1 0, E2 0, E3 0, E4 0 } C_DIS
LIN{ E6POS: X 782.3535, Y -67.5833, Z -90.0150, A 0, B 90, C 0, E1 0, E2 0, E3 0, E4 0 } C_DIS
LIN{ E6POS: X 782.1776, Y -68.5677, Z -90.0150, A 0, B 90, C 0, E1 0, E2 0, E3 0, E4 0 } C_DIS
LIN{ E6POS: X 782.0016, Y -69.5521, Z -90.0150, A 0, B 90, C 0, E1 0, E2 0, E3 0, E4 0 } C_DIS
LIN{ E6POS: X 781.8257, Y -70.5365, Z -90.0150, A 0, B 90, C 0, E1 0, E2 0, E3 0, E4 0 } C_DIS
LIN{ E6POS: X 781.7943, Y -70.7119, Z -90.0150, A 0, B 90, C 0, E1 0, E2 0, E3 0, E4 0 } C_DIS
LIN{ E6POS: X 781.5865, Y -71.6900, Z -90.0150, A 0, B 90, C 0, E1 0, E2 0, E3 0, E4 0 } C_DIS
LIN{ E6POS: X 781.3787, Y -72.6682, Z -90.0150, A 0, B 90, C 0, E1 0, E2 0, E3 0, E4 0 } C_DIS
LIN{ E6POS: X 781.1709, Y -73.6464, Z -90.0150, A 0, B 90, C 0, E1 0, E2 0, E3 0, E4 0 } C_DIS
LIN{ E6POS: X 780.9631, Y -74.6245, Z -90.0150, A 0, B 90, C 0, E1 0, E2 0, E3 0, E4 0 } C_DIS
LIN{ E6POS: X 780.7553, Y -75.6027, Z -90.0150, A 0, B 90, C 0, E1 0, E2 0, E3 0, E4 0 } C_DIS
LIN{ E6POS: X 780.5475, Y -76.5809, Z -90.0150, A 0, B 90, C 0, E1 0, E2 0, E3 0, E4 0 } C_DIS
LIN{ E6POS: X 780.3397, Y -77.5590, Z -90.0150, A 0, B 90, C 0, E1 0, E2 0, E3 0, E4 0 } C_DIS
LIN{ E6POS: X 780.2638, Y -77.9163, Z -90.0150, A 0, B 90, C 0, E1 0, E2 0, E3 0, E4 0 } C_DIS
LIN{ E6POS: X 780.0560, Y -78.8945, Z -90.0150, A 0, B 90, C 0, E1 0, E2 0, E3 0, E4 0 } C_DIS
LIN{ E6POS: X 779.8482, Y -79.8727, Z -90.0150, A 0, B 90, C 0, E1 0, E2 0, E3 0, E4 0 } C_DIS
LIN{ E6POS: X 779.6404, Y -80.8508, Z -90.0150, A 0, B 90, C 0, E1 0, E2 0, E3 0, E4 0 } C_DIS
LIN{ E6POS: X 779.4326, Y -81.8290, Z -90.0150, A 0, B 90, C 0, E1 0, E2 0, E3 0, E4 0 } C_DIS
LIN{ E6POS: X 779.2248, Y -82.8072, Z -90.0150, A 0, B 90, C 0, E1 0, E2 0, E3 0, E4 0 } C_DIS
LIN{ E6POS: X 779.0170, Y -83.7854, Z -90.0150, A 0, B 90, C 0, E1 0, E2 0, E3 0, E4 0 } C_DIS
LIN{ E6POS: X 778.8092, Y -84.7635, Z -90.0150, A 0, B 90, C 0, E1 0, E2 0, E3 0, E4 0 } C_DIS
LIN{ E6POS: X 778.6014, Y -85.7417, Z -90.0150, A 0, B 90, C 0, E1 0, E2 0, E3 0, E4 0 } C_DIS
LIN{ E6POS: X 778.3936, Y -86.7199, Z -90.0150, A 0, B 90, C 0, E1 0, E2 0, E3 0, E4 0 } C_DIS
LIN{ E6POS: X 778.1858, Y -87.6980, Z -90.0150, A 0, B 90, C 0, E1 0, E2 0, E3 0, E4 0 } C_DIS
LIN{ E6POS: X 777.9780, Y -88.6762, Z -90.0150, A 0, B 90, C 0, E1 0, E2 0, E3 0, E4 0 } C_DIS
LIN{ E6POS: X 777.7702, Y -89.6544, Z -90.0150, A 0, B 90, C 0, E1 0, E2 0, E3 0, E4 0 } C_DIS
LIN{ E6POS: X 777.5624, Y -90.6326, Z -90.0150, A 0, B 90, C 0, E1 0, E2 0, E3 0, E4 0 } C_DIS
LIN{ E6POS: X 777.5429, Y -90.7243, Z -90.0150, A 0, B 90, C 0, E1 0, E2 0, E3 0, E4 0 } C_DIS
LIN{ E6POS: X 777.3226, Y -91.6997, Z -90.0150, A 0, B 90, C 0, E1 0, E2 0, E3 0, E4 0 } C_DIS
LIN{ E6POS: X 777.1022, Y -92.6751, Z -90.0150, A 0, B 90, C 0, E1 0, E2 0, E3 0, E4 0 } C_DIS
LIN{ E6POS: X 776.8819, Y -93.6506, Z -90.0150, A 0, B 90, C 0, E1 0, E2 0, E3 0, E4 0 } C_DIS
LIN{ E6POS: X 776.6615, Y -94.6260, Z -90.0150, A 0, B 90, C 0, E1 0, E2 0, E3 0, E4 0 } C_DIS
LIN{ E6POS: X 776.4412, Y -95.6014, Z -90.0150, A 0, B 90, C 0, E1 0, E2 0, E3 0, E4 0 } C_DIS
LIN{ E6POS: X 776.2208, Y -96.5768, Z -90.0150, A 0, B 90, C 0, E1 0, E2 0, E3 0, E4 0 } C_DIS
LIN{ E6POS: X 776.0005, Y -97.5522, Z -90.0150, A 0, B 90, C 0, E1 0, E2 0, E3 0, E4 0 } C_DIS
LIN{ E6POS: X 775.8008, Y -98.4362, Z -90.0150, A 0, B 90, C 0, E1 0, E2 0, E3 0, E4 0 } C_DIS
LIN{ E6POS: X 775.5805, Y -99.4116, Z -90.0150, A 0, B 90, C 0, E1 0, E2 0, E3 0, E4 0 } C_DIS
LIN{ E6POS: X 775.3601, Y -100.3870, Z -90.0150, A 0, B 90, C 0, E1 0, E2 0, E3 0, E4 0 } C_DIS
LIN{ E6POS: X 775.1398, Y -101.3624, Z -90.0150, A 0, B 90, C 0, E1 0, E2 0, E3 0, E4 0 } C_DIS
LIN{ E6POS: X 774.9194, Y -102.3379, Z -90.0150, A 0, B 90, C 0, E1 0, E2 0, E3 0, E4 0 } C_DIS
LIN{ E6POS: X 774.6991, Y -103.3133, Z -90.0150, A 0, B 90, C 0, E1 0, E2 0, E3 0, E4 0 } C_DIS
LIN{ E6POS: X 774.4787, Y -104.2887, Z -90.0150, A 0, B 90, C 0, E1 0, E2 0, E3 0, E4 0 } C_DIS
LIN{ E6POS: X 774.2584, Y -105.2641, Z -90.0150, A 0, B 90, C 0, E1 0, E2 0, E3 0, E4 0 } C_DIS
LIN{ E6POS: X 774.0381, Y -106.2396, Z -90.0150, A 0, B 90, C 0, E1 0, E2 0, E3 0, E4 0 } C_DIS
LIN{ E6POS: X 773.8177, Y -107.2150, Z -90.0150, A 0, B 90, C 0, E1 0, E2 0, E3 0, E4 0 } C_DIS
LIN{ E6POS: X 773.5974, Y -108.1904, Z -90.0150, A 0, B 90, C 0, E1 0, E2 0, E3 0, E4 0 } C_DIS
LIN{ E6POS: X 773.3770, Y -109.1658, Z -90.0150, A 0, B 90, C 0, E1 0, E2 0, E3 0, E4 0 } C_DIS
LIN{ E6POS: X 773.1567, Y -110.1412, Z -90.0150, A 0, B 90, C 0, E1 0, E2 0, E3 0, E4 0 } C_DIS
LIN{ E6POS: X 772.9363, Y -111.1167, Z -90.0150, A 0, B 90, C 0, E1 0, E2 0, E3 0, E4 0 } C_DIS
LIN{ E6POS: X 772.7160, Y -112.0921, Z -90.0150, A 0, B 90, C 0, E1 0, E2 0, E3 0, E4 0 } C_DIS
LIN{ E6POS: X 772.7038, Y -112.1462, Z -90.0150, A 0, B 90, C 0, E1 0, E2 0, E3 0, E4 0 } C_DIS
LIN{ E6POS: X 772.0412, Y -111.3972, Z -90.0150, A 0, B 90, C 0, E1 0, E2 0, E3 0, E4 0 } C_DIS
LIN{ E6POS: X 771.7418, Y -111.0586, Z -90.0150, A 0, B 90, C 0, E1 0, E2 0, E3 0, E4 0 } C_DIS
LIN{ E6POS: X 771.0792, Y -110.3095, Z -90.0150, A 0, B 90, C 0, E1 0, E2 0, E3 0, E4 0 } C_DIS
LIN{ E6POS: X 770.4167, Y -109.5605, Z -90.0150, A 0, B 90, C 0, E1 0, E2 0, E3 0, E4 0 } C_DIS
LIN{ E6POS: X 770.0315, Y -109.1250, Z -90.0150, A 0, B 90, C 0, E1 0, E2 0, E3 0, E4 0 } C_DIS
LIN{ E6POS: X 769.2888, Y -108.4553, Z -90.0150, A 0, B 90, C 0, E1 0, E2 0, E3 0, E4 0 } C_DIS
LIN{ E6POS: X 768.7626, Y -107.9808, Z -90.0150, A 0, B 90, C 0, E1 0, E2 0, E3 0, E4 0 } C_DIS
LIN{ E6POS: X 768.0207, Y -107.3102, Z -90.0150, A 0, B 90, C 0, E1 0, E2 0, E3 0, E4 0 } C_DIS
LIN{ E6POS: X 767.2789, Y -106.6396, Z -90.0150, A 0, B 90, C 0, E1 0, E2 0, E3 0, E4 0 } C_DIS
LIN{ E6POS: X 766.5371, Y -105.9690, Z -90.0150, A 0, B 90, C 0, E1 0, E2 0, E3 0, E4 0 } C_DIS
LIN{ E6POS: X 766.5224, Y -105.9558, Z -90.0150, A 0, B 90, C 0, E1 0, E2 0, E3 0, E4 0 } C_DIS
LIN{ E6POS: X 765.6912, Y -105.3998, Z -90.0150, A 0, B 90, C 0, E1 0, E2 0, E3 0, E4 0 } C_DIS
LIN{ E6POS: X 764.8601, Y -104.8438, Z -90.0150, A 0, B 90, C 0, E1 0, E2 0, E3 0, E4 0 } C_DIS
LIN{ E6POS: X 764.0289, Y -104.2878, Z -90.0150, A 0, B 90, C 0, E1 0, E2 0, E3 0, E4 0 } C_DIS
LIN{ E6POS: X 763.2224, Y -103.7483, Z -90.0150, A 0, B 90, C 0, E1 0, E2 0, E3 0, E4 0 } C_DIS
LIN{ E6POS: X 762.3907, Y -103.1931, Z -90.0150, A 0, B 90, C 0, E1 0, E2 0, E3 0, E4 0 } C_DIS
LIN{ E6POS: X 761.5589, Y -102.6379, Z -90.0150, A 0, B 90, C 0, E1 0, E2 0, E3 0, E4 0 } C_DIS
LIN{ E6POS: X 761.3398, Y -102.4916, Z -90.0150, A 0, B 90, C 0, E1 0, E2 0, E3 0, E4 0 } C_DIS
LIN{ E6POS: X 760.4480, Y -102.0391, Z -90.0150, A 0, B 90, C 0, E1 0, E2 0, E3 0, E4 0 } C_DIS
LIN{ E6POS: X 759.5563, Y -101.5866, Z -90.0150, A 0, B 90, C 0, E1 0, E2 0, E3 0, E4 0 } C_DIS
LIN{ E6POS: X 758.6645, Y -101.1340, Z -90.0150, A 0, B 90, C 0, E1 0, E2 0, E3 0, E4 0 } C_DIS
LIN{ E6POS: X 757.7728, Y -100.6815, Z -90.0150, A 0, B 90, C 0, E1 0, E2 0, E3 0, E4 0 } C_DIS
LIN{ E6POS: X 756.8810, Y -100.2290, Z -90.0150, A 0, B 90, C 0, E1 0, E2 0, E3 0, E4 0 } C_DIS
LIN{ E6POS: X 756.4505, Y -100.0105, Z -90.0150, A 0, B 90, C 0, E1 0, E2 0, E3 0, E4 0 } C_DIS
LIN{ E6POS: X 755.5592, Y -99.5569, Z -90.0150, A 0, B 90, C 0, E1 0, E2 0, E3 0, E4 0 } C_DIS
LIN{ E6POS: X 754.6680, Y -99.1034, Z -90.0150, A 0, B 90, C 0, E1 0, E2 0, E3 0, E4 0 } C_DIS
LIN{ E6POS: X 753.7768, Y -98.6499, Z -90.0150, A 0, B 90, C 0, E1 0, E2 0, E3 0, E4 0 } C_DIS
LIN{ E6POS: X 753.6475, Y -98.5841, Z -90.0150, A 0, B 90, C 0, E1 0, E2 0, E3 0, E4 0 } C_DIS
LIN{ E6POS: X 752.7209, Y -98.2078, Z -90.0150, A 0, B 90, C 0, E1 0, E2 0, E3 0, E4 0 } C_DIS
LIN{ E6POS: X 751.7944, Y -97.8315, Z -90.0150, A 0, B 90, C 0, E1 0, E2 0, E3 0, E4 0 } C_DIS
LIN{ E6POS: X 750.8679, Y -97.4552, Z -90.0150, A 0, B 90, C 0, E1 0, E2 0, E3 0, E4 0 } C_DIS
LIN{ E6POS: X 749.9414, Y -97.0790, Z -90.0150, A 0, B 90, C 0, E1 0, E2 0, E3 0, E4 0 } C_DIS
LIN{ E6POS: X 749.0149, Y -96.7027, Z -90.0150, A 0, B 90, C 0, E1 0, E2 0, E3 0, E4 0 } C_DIS
LIN{ E6POS: X 748.0884, Y -96.3264, Z -90.0150, A 0, B 90, C 0, E1 0, E2 0, E3 0, E4 0 } C_DIS
LIN{ E6POS: X 747.1619, Y -95.9501, Z -90.0150, A 0, B 90, C 0, E1 0, E2 0, E3 0, E4 0 } C_DIS
LIN{ E6POS: X 746.6385, Y -95.7375, Z -90.0150, A 0, B 90, C 0, E1 0, E2 0, E3 0, E4 0 } C_DIS
LIN{ E6POS: X 745.7131, Y -95.3584, Z -90.0150, A 0, B 90, C 0, E1 0, E2 0, E3 0, E4 0 } C_DIS
LIN{ E6POS: X 744.7878, Y -94.9792, Z -90.0150, A 0, B 90, C 0, E1 0, E2 0, E3 0, E4 0 } C_DIS
LIN{ E6POS: X 743.8625, Y -94.6000, Z -90.0150, A 0, B 90, C 0, E1 0, E2 0, E3 0, E4 0 } C_DIS
LIN{ E6POS: X 742.9371, Y -94.2209, Z -90.0150, A 0, B 90, C 0, E1 0, E2 0, E3 0, E4 0 } C_DIS
LIN{ E6POS: X 742.6081, Y -94.0861, Z -90.0150, A 0, B 90, C 0, E1 0, E2 0, E3 0, E4 0 } C_DIS
LIN{ E6POS: X 741.6691, Y -93.7423, Z -90.0150, A 0, B 90, C 0, E1 0, E2 0, E3 0, E4 0 } C_DIS
LIN{ E6POS: X 740.7300, Y -93.3986, Z -90.0150, A 0, B 90, C 0, E1 0, E2 0, E3 0, E4 0 } C_DIS
LIN{ E6POS: X 739.7909, Y -93.0548, Z -90.0150, A 0, B 90, C 0, E1 0, E2 0, E3 0, E4 0 } C_DIS
LIN{ E6POS: X 738.8519, Y -92.7111, Z -90.0150, A 0, B 90, C 0, E1 0, E2 0, E3 0, E4 0 } C_DIS
LIN{ E6POS: X 737.9128, Y -92.3674, Z -90.0150, A 0, B 90, C 0, E1 0, E2 0, E3 0, E4 0 } C_DIS
LIN{ E6POS: X 736.9737, Y -92.0236, Z -90.0150, A 0, B 90, C 0, E1 0, E2 0, E3 0, E4 0 } C_DIS
LIN{ E6POS: X 736.0347, Y -91.6799, Z -90.0150, A 0, B 90, C 0, E1 0, E2 0, E3 0, E4 0 } C_DIS
LIN{ E6POS: X 735.0956, Y -91.3362, Z -90.0150, A 0, B 90, C 0, E1 0, E2 0, E3 0, E4 0 } C_DIS
LIN{ E6POS: X 734.6493, Y -91.1728, Z -90.0150, A 0, B 90, C 0, E1 0, E2 0, E3 0, E4 0 } C_DIS
LIN{ E6POS: X 733.7115, Y -90.8257, Z -90.0150, A 0, B 90, C 0, E1 0, E2 0, E3 0, E4 0 } C_DIS
LIN{ E6POS: X 732.7737, Y -90.4786, Z -90.0150, A 0, B 90, C 0, E1 0, E2 0, E3 0, E4 0 } C_DIS
LIN{ E6POS: X 731.8358, Y -90.1315, Z -90.0150, A 0, B 90, C 0, E1 0, E2 0, E3 0, E4 0 } C_DIS
LIN{ E6POS: X 730.8980, Y -89.7844, Z -90.0150, A 0, B 90, C 0, E1 0, E2 0, E3 0, E4 0 } C_DIS
LIN{ E6POS: X 730.0656, Y -89.4763, Z -90.0150, A 0, B 90, C 0, E1 0, E2 0, E3 0, E4 0 } C_DIS
LIN{ E6POS: X 729.1208, Y -89.1487, Z -90.0150, A 0, B 90, C 0, E1 0, E2 0, E3 0, E4 0 } C_DIS
LIN{ E6POS: X 728.1760, Y -88.8211, Z -90.0150, A 0, B 90, C 0, E1 0, E2 0, E3 0, E4 0 } C_DIS
LIN{ E6POS: X 727.2312, Y -88.4935, Z -90.0150, A 0, B 90, C 0, E1 0, E2 0, E3 0, E4 0 } C_DIS
LIN{ E6POS: X 726.2863, Y -88.1659, Z -90.0150, A 0, B 90, C 0, E1 0, E2 0, E3 0, E4 0 } C_DIS
LIN{ E6POS: X 725.3415, Y -87.8383, Z -90.0150, A 0, B 90, C 0, E1 0, E2 0, E3 0, E4 0 } C_DIS
LIN{ E6POS: X 724.3967, Y -87.5107, Z -90.0150, A 0, B 90, C 0, E1 0, E2 0, E3 0, E4 0 } C_DIS
LIN{ E6POS: X 723.4519, Y -87.1832, Z -90.0150, A 0, B 90, C 0, E1 0, E2 0, E3 0, E4 0 } C_DIS
LIN{ E6POS: X 722.5071, Y -86.8556, Z -90.0150, A 0, B 90, C 0, E1 0, E2 0, E3 0, E4 0 } C_DIS
LIN{ E6POS: X 722.3251, Y -86.7925, Z -90.0150, A 0, B 90, C 0, E1 0, E2 0, E3 0, E4 0 } C_DIS
LIN{ E6POS: X 721.3811, Y -86.4624, Z -90.0150, A 0, B 90, C 0, E1 0, E2 0, E3 0, E4 0 } C_DIS
LIN{ E6POS: X 720.4372, Y -86.1323, Z -90.0150, A 0, B 90, C 0, E1 0, E2 0, E3 0, E4 0 } C_DIS
LIN{ E6POS: X 719.4932, Y -85.8022, Z -90.0150, A 0, B 90, C 0, E1 0, E2 0, E3 0, E4 0 } C_DIS
LIN{ E6POS: X 718.5493, Y -85.4721, Z -90.0150, A 0, B 90, C 0, E1 0, E2 0, E3 0, E4 0 } C_DIS
LIN{ E6POS: X 717.8615, Y -85.2316, Z -90.0150, A 0, B 90, C 0, E1 0, E2 0, E3 0, E4 0 } C_DIS
LIN{ E6POS: X 716.9145, Y -84.9104, Z -90.0150, A 0, B 90, C 0, E1 0, E2 0, E3 0, E4 0 } C_DIS
LIN{ E6POS: X 715.9674, Y -84.5893, Z -90.0150, A 0, B 90, C 0, E1 0, E2 0, E3 0, E4 0 } C_DIS
LIN{ E6POS: X 715.0204, Y -84.2681, Z -90.0150, A 0, B 90, C 0, E1 0, E2 0, E3 0, E4 0 } C_DIS
LIN{ E6POS: X 714.0734, Y -83.9469, Z -90.0150, A 0, B 90, C 0, E1 0, E2 0, E3 0, E4 0 } C_DIS
LIN{ E6POS: X 713.1264, Y -83.6257, Z -90.0150, A 0, B 90, C 0, E1 0, E2 0, E3 0, E4 0 } C_DIS
LIN{ E6POS: X 712.1794, Y -83.3045, Z -90.0150, A 0, B 90, C 0, E1 0, E2 0, E3 0, E4 0 } C_DIS
LIN{ E6POS: X 711.5083, Y -83.0769, Z -90.0150, A 0, B 90, C 0, E1 0, E2 0, E3 0, E4 0 } C_DIS
LIN{ E6POS: X 710.5612, Y -82.7559, Z -90.0150, A 0, B 90, C 0, E1 0, E2 0, E3 0, E4 0 } C_DIS
LIN{ E6POS: X 709.6141, Y -82.4350, Z -90.0150, A 0, B 90, C 0, E1 0, E2 0, E3 0, E4 0 } C_DIS
LIN{ E6POS: X 708.6670, Y -82.1140, Z -90.0150, A 0, B 90, C 0, E1 0, E2 0, E3 0, E4 0 } C_DIS
LIN{ E6POS: X 707.8389, Y -81.8334, Z -90.0150, A 0, B 90, C 0, E1 0, E2 0, E3 0, E4 0 } C_DIS
LIN{ E6POS: X 706.8951, Y -81.5029, Z -90.0150, A 0, B 90, C 0, E1 0, E2 0, E3 0, E4 0 } C_DIS
LIN{ E6POS: X 705.9512, Y -81.1725, Z -90.0150, A 0, B 90, C 0, E1 0, E2 0, E3 0, E4 0 } C_DIS
LIN{ E6POS: X 705.0074, Y -80.8421, Z -90.0150, A 0, B 90, C 0, E1 0, E2 0, E3 0, E4 0 } C_DIS
LIN{ E6POS: X 704.0636, Y -80.5116, Z -90.0150, A 0, B 90, C 0, E1 0, E2 0, E3 0, E4 0 } C_DIS
LIN{ E6POS: X 704.0428, Y -80.5044, Z -90.0150, A 0, B 90, C 0, E1 0, E2 0, E3 0, E4 0 } C_DIS
LIN{ E6POS: X 703.0957, Y -80.1834, Z -90.0150, A 0, B 90, C 0, E1 0, E2 0, E3 0, E4 0 } C_DIS
LIN{ E6POS: X 702.1486, Y -79.8623, Z -90.0150, A 0, B 90, C 0, E1 0, E2 0, E3 0, E4 0 } C_DIS
LIN{ E6POS: X 701.8410, Y -79.7581, Z -90.0150, A 0, B 90, C 0, E1 0, E2 0, E3 0, E4 0 } C_DIS
LIN{ E6POS: X 700.9055, Y -79.4047, Z -90.0150, A 0, B 90, C 0, E1 0, E2 0, E3 0, E4 0 } C_DIS
LIN{ E6POS: X 699.9701, Y -79.0513, Z -90.0150, A 0, B 90, C 0, E1 0, E2 0, E3 0, E4 0 } C_DIS
LIN{ E6POS: X 699.9619, Y -79.0483, Z -90.0150, A 0, B 90, C 0, E1 0, E2 0, E3 0, E4 0 } C_DIS
LIN{ E6POS: X 699.0148, Y -78.7271, Z -90.0150, A 0, B 90, C 0, E1 0, E2 0, E3 0, E4 0 } C_DIS
LIN{ E6POS: X 698.8609, Y -78.6749, Z -90.0150, A 0, B 90, C 0, E1 0, E2 0, E3 0, E4 0 } C_DIS
LIN{ E6POS: X 698.2865, Y -78.3180, Z -90.0150, A 0, B 90, C 0, E1 0, E2 0, E3 0, E4 0 } C_DIS
LIN{ E6POS: X 697.9197, Y -78.1937, Z -90.0150, A 0, B 90, C 0, E1 0, E2 0, E3 0, E4 0 } C_DIS
LIN{ E6POS: X 697.9888, Y -77.7446, Z -90.0150, A 0, B 90, C 0, E1 0, E2 0, E3 0, E4 0 } C_DIS
LIN{ E6POS: X 698.1681, Y -76.8647, Z -90.0150, A 0, B 90, C 0, E1 0, E2 0, E3 0, E4 0 } C_DIS
LIN{ E6POS: X 698.2408, Y -76.4081, Z -90.0150, A 0, B 90, C 0, E1 0, E2 0, E3 0, E4 0 } C_DIS
LIN{ E6POS: X 698.4116, Y -75.5521, Z -90.0150, A 0, B 90, C 0, E1 0, E2 0, E3 0, E4 0 } C_DIS
LIN{ E6POS: X 698.4918, Y -75.0807, Z -90.0150, A 0, B 90, C 0, E1 0, E2 0, E3 0, E4 0 } C_DIS
LIN{ E6POS: X 698.6720, Y -74.2137, Z -90.0150, A 0, B 90, C 0, E1 0, E2 0, E3 0, E4 0 } C_DIS
LIN{ E6POS: X 698.7632, Y -73.7198, Z -90.0150, A 0, B 90, C 0, E1 0, E2 0, E3 0, E4 0 } C_DIS
LIN{ E6POS: X 698.9564, Y -72.8350, Z -90.0150, A 0, B 90, C 0, E1 0, E2 0, E3 0, E4 0 } C_DIS
LIN{ E6POS: X 699.0622, Y -72.3117, Z -90.0150, A 0, B 90, C 0, E1 0, E2 0, E3 0, E4 0 } C_DIS
LIN{ E6POS: X 699.2734, Y -71.4039, Z -90.0150, A 0, B 90, C 0, E1 0, E2 0, E3 0, E4 0 } C_DIS
LIN{ E6POS: X 699.3888, Y -70.8581, Z -90.0150, A 0, B 90, C 0, E1 0, E2 0, E3 0, E4 0 } C_DIS
LIN{ E6POS: X 699.6109, Y -69.9290, Z -90.0150, A 0, B 90, C 0, E1 0, E2 0, E3 0, E4 0 } C_DIS
LIN{ E6POS: X 699.7293, Y -69.3685, Z -90.0150, A 0, B 90, C 0, E1 0, E2 0, E3 0, E4 0 } C_DIS
LIN{ E6POS: X 699.9542, Y -68.4191, Z -90.0150, A 0, B 90, C 0, E1 0, E2 0, E3 0, E4 0 } C_DIS
LIN{ E6POS: X 700.0706, Y -67.8508, Z -90.0150, A 0, B 90, C 0, E1 0, E2 0, E3 0, E4 0 } C_DIS
LIN{ E6POS: X 700.2910, Y -66.8840, Z -90.0150, A 0, B 90, C 0, E1 0, E2 0, E3 0, E4 0 } C_DIS
LIN{ E6POS: X 700.4000, Y -66.3153, Z -90.0150, A 0, B 90, C 0, E1 0, E2 0, E3 0, E4 0 } C_DIS
LIN{ E6POS: X 700.6067, Y -65.3369, Z -90.0150, A 0, B 90, C 0, E1 0, E2 0, E3 0, E4 0 } C_DIS
LIN{ E6POS: X 700.6079, Y -65.3312, Z -90.0150, A 0, B 90, C 0, E1 0, E2 0, E3 0, E4 0 } C_DIS
LIN{ E6POS: X 700.7075, Y -64.7700, Z -90.0150, A 0, B 90, C 0, E1 0, E2 0, E3 0, E4 0 } C_DIS
LIN{ E6POS: X 700.9020, Y -63.7891, Z -90.0150, A 0, B 90, C 0, E1 0, E2 0, E3 0, E4 0 } C_DIS
LIN{ E6POS: X 700.9023, Y -63.7879, Z -90.0150, A 0, B 90, C 0, E1 0, E2 0, E3 0, E4 0 } C_DIS
LIN{ E6POS: X 700.9920, Y -63.2415, Z -90.0150, A 0, B 90, C 0, E1 0, E2 0, E3 0, E4 0 } C_DIS
LIN{ E6POS: X 701.1716, Y -62.2786, Z -90.0150, A 0, B 90, C 0, E1 0, E2 0, E3 0, E4 0 } C_DIS
LIN{ E6POS: X 701.2490, Y -61.7546, Z -90.0150, A 0, B 90, C 0, E1 0, E2 0, E3 0, E4 0 } C_DIS
LIN{ E6POS: X 701.4120, Y -60.8304, Z -90.0150, A 0, B 90, C 0, E1 0, E2 0, E3 0, E4 0 } C_DIS
LIN{ E6POS: X 701.4767, Y -60.3364, Z -90.0150, A 0, B 90, C 0, E1 0, E2 0, E3 0, E4 0 } C_DIS
LIN{ E6POS: X 701.6216, Y -59.4684, Z -90.0150, A 0, B 90, C 0, E1 0, E2 0, E3 0, E4 0 } C_DIS
LIN{ E6POS: X 701.6784, Y -58.9896, Z -90.0150, A 0, B 90, C 0, E1 0, E2 0, E3 0, E4 0 } C_DIS
LIN{ E6POS: X 701.8112, Y -58.1497, Z -90.0150, A 0, B 90, C 0, E1 0, E2 0, E3 0, E4 0 } C_DIS
LIN{ E6POS: X 701.9380, Y -57.3099, Z -90.0150, A 0, B 90, C 0, E1 0, E2 0, E3 0, E4 0 } C_DIS
LIN{ E6POS: X 701.9911, Y -56.8307, Z -90.0150, A 0, B 90, C 0, E1 0, E2 0, E3 0, E4 0 } C_DIS
LIN{ E6POS: X 702.1184, Y -55.9631, Z -90.0150, A 0, B 90, C 0, E1 0, E2 0, E3 0, E4 0 } C_DIS
LIN{ E6POS: X 702.1732, Y -55.4695, Z -90.0150, A 0, B 90, C 0, E1 0, E2 0, E3 0, E4 0 } C_DIS
LIN{ E6POS: X 702.3067, Y -54.5453, Z -90.0150, A 0, B 90, C 0, E1 0, E2 0, E3 0, E4 0 } C_DIS
LIN{ E6POS: X 702.3679, Y -54.0211, Z -90.0150, A 0, B 90, C 0, E1 0, E2 0, E3 0, E4 0 } C_DIS
LIN{ E6POS: X 702.5024, Y -53.0693, Z -90.0150, A 0, B 90, C 0, E1 0, E2 0, E3 0, E4 0 } C_DIS
LIN{ E6POS: X 702.5657, Y -52.5308, Z -90.0150, A 0, B 90, C 0, E1 0, E2 0, E3 0, E4 0 } C_DIS
LIN{ E6POS: X 702.6953, Y -51.5794, Z -90.0150, A 0, B 90, C 0, E1 0, E2 0, E3 0, E4 0 } C_DIS
LIN{ E6POS: X 702.7559, Y -51.0408, Z -90.0150, A 0, B 90, C 0, E1 0, E2 0, E3 0, E4 0 } C_DIS
LIN{ E6POS: X 702.8758, Y -50.1177, Z -90.0150, A 0, B 90, C 0, E1 0, E2 0, E3 0, E4 0 } C_DIS
LIN{ E6POS: X 702.9294, Y -49.5941, Z -90.0150, A 0, B 90, C 0, E1 0, E2 0, E3 0, E4 0 } C_DIS
LIN{ E6POS: X 703.0342, Y -48.7275, Z -90.0150, A 0, B 90, C 0, E1 0, E2 0, E3 0, E4 0 } C_DIS
LIN{ E6POS: X 703.0763, Y -48.2343, Z -90.0150, A 0, B 90, C 0, E1 0, E2 0, E3 0, E4 0 } C_DIS
LIN{ E6POS: X 703.1672, Y -47.4379, Z -90.0150, A 0, B 90, C 0, E1 0, E2 0, E3 0, E4 0 } C_DIS
LIN{ E6POS: X 703.1995, Y -46.9880, Z -90.0150, A 0, B 90, C 0, E1 0, E2 0, E3 0, E4 0 } C_DIS
LIN{ E6POS: X 703.3198, Y -45.9953, Z -90.0150, A 0, B 90, C 0, E1 0, E2 0, E3 0, E4 0 } C_DIS
LIN{ E6POS: X 703.4401, Y -45.0026, Z -90.0150, A 0, B 90, C 0, E1 0, E2 0, E3 0, E4 0 } C_DIS
LIN{ E6POS: X 703.4454, Y -44.9588, Z -90.0150, A 0, B 90, C 0, E1 0, E2 0, E3 0, E4 0 } C_DIS
LIN{ E6POS: X 703.5123, Y -43.9610, Z -90.0150, A 0, B 90, C 0, E1 0, E2 0, E3 0, E4 0 } C_DIS
LIN{ E6POS: X 703.5228, Y -43.8038, Z -90.0150, A 0, B 90, C 0, E1 0, E2 0, E3 0, E4 0 } C_DIS
LIN{ E6POS: X 703.6468, Y -42.8116, Z -90.0150, A 0, B 90, C 0, E1 0, E2 0, E3 0, E4 0 } C_DIS
LIN{ E6POS: X 703.7609, Y -41.8985, Z -90.0150, A 0, B 90, C 0, E1 0, E2 0, E3 0, E4 0 } C_DIS
LIN{ E6POS: X 703.8412, Y -40.9018, Z -90.0150, A 0, B 90, C 0, E1 0, E2 0, E3 0, E4 0 } C_DIS
LIN{ E6POS: X 703.8539, Y -40.7436, Z -90.0150, A 0, B 90, C 0, E1 0, E2 0, E3 0, E4 0 } C_DIS
LIN{ E6POS: X 703.9344, Y -39.9924, Z -90.0150, A 0, B 90, C 0, E1 0, E2 0, E3 0, E4 0 } C_DIS
LIN{ E6POS: X 703.9659, Y -39.5615, Z -90.0150, A 0, B 90, C 0, E1 0, E2 0, E3 0, E4 0 } C_DIS
LIN{ E6POS: X 704.0456, Y -38.7548, Z -90.0150, A 0, B 90, C 0, E1 0, E2 0, E3 0, E4 0 } C_DIS
LIN{ E6POS: X 704.0730, Y -38.3042, Z -90.0150, A 0, B 90, C 0, E1 0, E2 0, E3 0, E4 0 } C_DIS
LIN{ E6POS: X 704.1465, Y -37.4797, Z -90.0150, A 0, B 90, C 0, E1 0, E2 0, E3 0, E4 0 } C_DIS
LIN{ E6POS: X 704.1660, Y -37.0307, Z -90.0150, A 0, B 90, C 0, E1 0, E2 0, E3 0, E4 0 } C_DIS
LIN{ E6POS: X 704.2281, Y -36.2246, Z -90.0150, A 0, B 90, C 0, E1 0, E2 0, E3 0, E4 0 } C_DIS
LIN{ E6POS: X 704.2434, Y -35.7698, Z -90.0150, A 0, B 90, C 0, E1 0, E2 0, E3 0, E4 0 } C_DIS
LIN{ E6POS: X 704.2983, Y -34.9634, Z -90.0150, A 0, B 90, C 0, E1 0, E2 0, E3 0, E4 0 } C_DIS
LIN{ E6POS: X 704.3128, Y -34.4945, Z -90.0150, A 0, B 90, C 0, E1 0, E2 0, E3 0, E4 0 } C_DIS
LIN{ E6POS: X 704.3657, Y -33.6702, Z -90.0150, A 0, B 90, C 0, E1 0, E2 0, E3 0, E4 0 } C_DIS
LIN{ E6POS: X 704.3821, Y -33.1791, Z -90.0150, A 0, B 90, C 0, E1 0, E2 0, E3 0, E4 0 } C_DIS
LIN{ E6POS: X 704.4374, Y -32.3176, Z -90.0150, A 0, B 90, C 0, E1 0, E2 0, E3 0, E4 0 } C_DIS
LIN{ E6POS: X 704.4599, Y -31.7966, Z -90.0150, A 0, B 90, C 0, E1 0, E2 0, E3 0, E4 0 } C_DIS
LIN{ E6POS: X 704.5211, Y -30.8790, Z -90.0150, A 0, B 90, C 0, E1 0, E2 0, E3 0, E4 0 } C_DIS
LIN{ E6POS: X 704.5454, Y -30.3429, Z -90.0150, A 0, B 90, C 0, E1 0, E2 0, E3 0, E4 0 } C_DIS
LIN{ E6POS: X 704.6088, Y -29.3981, Z -90.0150, A 0, B 90, C 0, E1 0, E2 0, E3 0, E4 0 } C_DIS
LIN{ E6POS: X 704.6316, Y -28.8626, Z -90.0150, A 0, B 90, C 0, E1 0, E2 0, E3 0, E4 0 } C_DIS
LIN{ E6POS: X 704.6920, Y -27.9175, Z -90.0150, A 0, B 90, C 0, E1 0, E2 0, E3 0, E4 0 } C_DIS
LIN{ E6POS: X 704.7095, Y -27.3976, Z -90.0150, A 0, B 90, C 0, E1 0, E2 0, E3 0, E4 0 } C_DIS
LIN{ E6POS: X 704.7623, Y -26.4821, Z -90.0150, A 0, B 90, C 0, E1 0, E2 0, E3 0, E4 0 } C_DIS
LIN{ E6POS: X 704.7708, Y -25.9930, Z -90.0150, A 0, B 90, C 0, E1 0, E2 0, E3 0, E4 0 } C_DIS
LIN{ E6POS: X 704.8115, Y -25.1342, Z -90.0150, A 0, B 90, C 0, E1 0, E2 0, E3 0, E4 0 } C_DIS
LIN{ E6POS: X 704.8145, Y -24.6610, Z -90.0150, A 0, B 90, C 0, E1 0, E2 0, E3 0, E4 0 } C_DIS
LIN{ E6POS: X 704.8473, Y -23.8350, Z -90.0150, A 0, B 90, C 0, E1 0, E2 0, E3 0, E4 0 } C_DIS
LIN{ E6POS: X 704.8486, Y -23.3620, Z -90.0150, A 0, B 90, C 0, E1 0, E2 0, E3 0, E4 0 } C_DIS
LIN{ E6POS: X 704.8779, Y -22.5429, Z -90.0150, A 0, B 90, C 0, E1 0, E2 0, E3 0, E4 0 } C_DIS
LIN{ E6POS: X 704.8814, Y -22.0549, Z -90.0150, A 0, B 90, C 0, E1 0, E2 0, E3 0, E4 0 } C_DIS
LIN{ E6POS: X 704.9114, Y -21.2187, Z -90.0150, A 0, B 90, C 0, E1 0, E2 0, E3 0, E4 0 } C_DIS
LIN{ E6POS: X 704.9202, Y -20.7005, Z -90.0150, A 0, B 90, C 0, E1 0, E2 0, E3 0, E4 0 } C_DIS
LIN{ E6POS: X 704.9546, Y -19.8218, Z -90.0150, A 0, B 90, C 0, E1 0, E2 0, E3 0, E4 0 } C_DIS
LIN{ E6POS: X 704.9680, Y -19.2808, Z -90.0150, A 0, B 90, C 0, E1 0, E2 0, E3 0, E4 0 } C_DIS
LIN{ E6POS: X 705.0058, Y -18.3698, Z -90.0150, A 0, B 90, C 0, E1 0, E2 0, E3 0, E4 0 } C_DIS
LIN{ E6POS: X 705.0217, Y -17.8135, Z -90.0150, A 0, B 90, C 0, E1 0, E2 0, E3 0, E4 0 } C_DIS
LIN{ E6POS: X 705.0624, Y -16.8822, Z -90.0150, A 0, B 90, C 0, E1 0, E2 0, E3 0, E4 0 } C_DIS
LIN{ E6POS: X 705.0754, Y -16.1816, Z -90.0150, A 0, B 90, C 0, E1 0, E2 0, E3 0, E4 0 } C_DIS
LIN{ E6POS: X 705.1164, Y -15.1824, Z -90.0150, A 0, B 90, C 0, E1 0, E2 0, E3 0, E4 0 } C_DIS
LIN{ E6POS: X 705.1279, Y -14.9021, Z -90.0150, A 0, B 90, C 0, E1 0, E2 0, E3 0, E4 0 } C_DIS
LIN{ E6POS: X 705.1034, Y -14.1272, Z -90.0150, A 0, B 90, C 0, E1 0, E2 0, E3 0, E4 0 } C_DIS
LIN{ E6POS: X 705.1190, Y -13.1273, Z -90.0150, A 0, B 90, C 0, E1 0, E2 0, E3 0, E4 0 } C_DIS
LIN{ E6POS: X 705.1263, Y -12.6601, Z -90.0150, A 0, B 90, C 0, E1 0, E2 0, E3 0, E4 0 } C_DIS
LIN{ E6POS: X 705.1171, Y -12.2265, Z -90.0150, A 0, B 90, C 0, E1 0, E2 0, E3 0, E4 0 } C_DIS
LIN{ E6POS: X 705.1272, Y -11.4632, Z -90.0150, A 0, B 90, C 0, E1 0, E2 0, E3 0, E4 0 } C_DIS
LIN{ E6POS: X 705.1209, Y -10.9789, Z -90.0150, A 0, B 90, C 0, E1 0, E2 0, E3 0, E4 0 } C_DIS
LIN{ E6POS: X 705.1357, Y -10.1293, Z -90.0150, A 0, B 90, C 0, E1 0, E2 0, E3 0, E4 0 } C_DIS
LIN{ E6POS: X 705.1355, Y -9.6147, Z -90.0150, A 0, B 90, C 0, E1 0, E2 0, E3 0, E4 0 } C_DIS
LIN{ E6POS: X 705.1568, Y -8.7092, Z -90.0150, A 0, B 90, C 0, E1 0, E2 0, E3 0, E4 0 } C_DIS
LIN{ E6POS: X 705.1591, Y -8.1797, Z -90.0150, A 0, B 90, C 0, E1 0, E2 0, E3 0, E4 0 } C_DIS
LIN{ E6POS: X 705.1819, Y -7.2474, Z -90.0150, A 0, B 90, C 0, E1 0, E2 0, E3 0, E4 0 } C_DIS
LIN{ E6POS: X 705.1833, Y -6.7187, Z -90.0150, A 0, B 90, C 0, E1 0, E2 0, E3 0, E4 0 } C_DIS
LIN{ E6POS: X 705.2052, Y -5.7875, Z -90.0150, A 0, B 90, C 0, E1 0, E2 0, E3 0, E4 0 } C_DIS
LIN{ E6POS: X 705.2025, Y -5.2747, Z -90.0150, A 0, B 90, C 0, E1 0, E2 0, E3 0, E4 0 } C_DIS
LIN{ E6POS: X 705.2193, Y -4.3726, Z -90.0150, A 0, B 90, C 0, E1 0, E2 0, E3 0, E4 0 } C_DIS
LIN{ E6POS: X 705.2098, Y -3.8917, Z -90.0150, A 0, B 90, C 0, E1 0, E2 0, E3 0, E4 0 } C_DIS
LIN{ E6POS: X 705.2185, Y -3.0468, Z -90.0150, A 0, B 90, C 0, E1 0, E2 0, E3 0, E4 0 } C_DIS
LIN{ E6POS: X 705.2048, Y -2.5822, Z -90.0150, A 0, B 90, C 0, E1 0, E2 0, E3 0, E4 0 } C_DIS
LIN{ E6POS: X 705.2081, Y -1.7676, Z -90.0150, A 0, B 90, C 0, E1 0, E2 0, E3 0, E4 0 } C_DIS
LIN{ E6POS: X 705.1938, Y -1.3040, Z -90.0150, A 0, B 90, C 0, E1 0, E2 0, E3 0, E4 0 } C_DIS
LIN{ E6POS: X 705.1959, Y -0.4896, Z -90.0150, A 0, B 90, C 0, E1 0, E2 0, E3 0, E4 0 } C_DIS
LIN{ E6POS: X 705.1842, Y -0.0104, Z -90.0150, A 0, B 90, C 0, E1 0, E2 0, E3 0, E4 0 } C_DIS
LIN{ E6POS: X 705.1891, Y 0.8311, Z -90.0150, A 0, B 90, C 0, E1 0, E2 0, E3 0, E4 0 } C_DIS
LIN{ E6POS: X 705.1833, Y 1.3411, Z -90.0150, A 0, B 90, C 0, E1 0, E2 0, E3 0, E4 0 } C_DIS
LIN{ E6POS: X 705.1944, Y 2.2371, Z -90.0150, A 0, B 90, C 0, E1 0, E2 0, E3 0, E4 0 } C_DIS
LIN{ E6POS: X 705.1917, Y 2.7618, Z -90.0150, A 0, B 90, C 0, E1 0, E2 0, E3 0, E4 0 } C_DIS
LIN{ E6POS: X 705.2056, Y 3.6855, Z -90.0150, A 0, B 90, C 0, E1 0, E2 0, E3 0, E4 0 } C_DIS
LIN{ E6POS: X 705.2025, Y 4.2097, Z -90.0150, A 0, B 90, C 0, E1 0, E2 0, E3 0, E4 0 } C_DIS
LIN{ E6POS: X 705.2155, Y 5.1324, Z -90.0150, A 0, B 90, C 0, E1 0, E2 0, E3 0, E4 0 } C_DIS
LIN{ E6POS: X 705.2091, Y 5.6399, Z -90.0150, A 0, B 90, C 0, E1 0, E2 0, E3 0, E4 0 } C_DIS
LIN{ E6POS: X 705.2187, Y 6.5324, Z -90.0150, A 0, B 90, C 0, E1 0, E2 0, E3 0, E4 0 } C_DIS
LIN{ E6POS: X 705.2056, Y 7.0077, Z -90.0150, A 0, B 90, C 0, E1 0, E2 0, E3 0, E4 0 } C_DIS
LIN{ E6POS: X 705.2078, Y 7.8433, Z -90.0150, A 0, B 90, C 0, E1 0, E2 0, E3 0, E4 0 } C_DIS
LIN{ E6POS: X 705.2058, Y 8.6489, Z -90.0150, A 0, B 90, C 0, E1 0, E2 0, E3 0, E4 0 } C_DIS
LIN{ E6POS: X 705.1893, Y 9.1080, Z -90.0150, A 0, B 90, C 0, E1 0, E2 0, E3 0, E4 0 } C_DIS
LIN{ E6POS: X 705.1876, Y 9.9122, Z -90.0150, A 0, B 90, C 0, E1 0, E2 0, E3 0, E4 0 } C_DIS
LIN{ E6POS: X 705.1711, Y 10.3702, Z -90.0150, A 0, B 90, C 0, E1 0, E2 0, E3 0, E4 0 } C_DIS
LIN{ E6POS: X 705.1722, Y 11.2015, Z -90.0150, A 0, B 90, C 0, E1 0, E2 0, E3 0, E4 0 } C_DIS
LIN{ E6POS: X 705.1590, Y 11.6749, Z -90.0150, A 0, B 90, C 0, E1 0, E2 0, E3 0, E4 0 } C_DIS
LIN{ E6POS: X 705.1675, Y 12.5610, Z -90.0150, A 0, B 90, C 0, E1 0, E2 0, E3 0, E4 0 } C_DIS
LIN{ E6POS: X 705.1606, Y 13.0654, Z -90.0150, A 0, B 90, C 0, E1 0, E2 0, E3 0, E4 0 } C_DIS
LIN{ E6POS: X 705.1571, Y 13.5844, Z -90.0150, A 0, B 90, C 0, E1 0, E2 0, E3 0, E4 0 } C_DIS
LIN{ E6POS: X 705.1690, Y 14.4975, Z -90.0150, A 0, B 90, C 0, E1 0, E2 0, E3 0, E4 0 } C_DIS
LIN{ E6POS: X 705.1812, Y 15.4098, Z -90.0150, A 0, B 90, C 0, E1 0, E2 0, E3 0, E4 0 } C_DIS
LIN{ E6POS: X 705.1779, Y 15.9283, Z -90.0150, A 0, B 90, C 0, E1 0, E2 0, E3 0, E4 0 } C_DIS
LIN{ E6POS: X 705.1866, Y 16.8104, Z -90.0150, A 0, B 90, C 0, E1 0, E2 0, E3 0, E4 0 } C_DIS
LIN{ E6POS: X 705.1800, Y 17.3121, Z -90.0150, A 0, B 90, C 0, E1 0, E2 0, E3 0, E4 0 } C_DIS
LIN{ E6POS: X 705.1823, Y 18.1364, Z -90.0150, A 0, B 90, C 0, E1 0, E2 0, E3 0, E4 0 } C_DIS
LIN{ E6POS: X 705.1696, Y 18.6051, Z -90.0150, A 0, B 90, C 0, E1 0, E2 0, E3 0, E4 0 } C_DIS
LIN{ E6POS: X 705.1690, Y 19.3997, Z -90.0150, A 0, B 90, C 0, E1 0, E2 0, E3 0, E4 0 } C_DIS
LIN{ E6POS: X 705.1535, Y 19.8521, Z -90.0150, A 0, B 90, C 0, E1 0, E2 0, E3 0, E4 0 } C_DIS
LIN{ E6POS: X 705.1539, Y 20.6457, Z -90.0150, A 0, B 90, C 0, E1 0, E2 0, E3 0, E4 0 } C_DIS
LIN{ E6POS: X 705.1390, Y 21.0968, Z -90.0150, A 0, B 90, C 0, E1 0, E2 0, E3 0, E4 0 } C_DIS
LIN{ E6POS: X 705.1437, Y 21.9163, Z -90.0150, A 0, B 90, C 0, E1 0, E2 0, E3 0, E4 0 } C_DIS
LIN{ E6POS: X 705.1324, Y 22.3827, Z -90.0150, A 0, B 90, C 0, E1 0, E2 0, E3 0, E4 0 } C_DIS
LIN{ E6POS: X 705.1453, Y 23.2575, Z -90.0150, A 0, B 90, C 0, E1 0, E2 0, E3 0, E4 0 } C_DIS
LIN{ E6POS: X 705.1414, Y 23.7554, Z -90.0150, A 0, B 90, C 0, E1 0, E2 0, E3 0, E4 0 } C_DIS
LIN{ E6POS: X 705.1595, Y 24.6225, Z -90.0150, A 0, B 90, C 0, E1 0, E2 0, E3 0, E4 0 } C_DIS
LIN{ E6POS: X 705.1604, Y 25.1099, Z -90.0150, A 0, B 90, C 0, E1 0, E2 0, E3 0, E4 0 } C_DIS
LIN{ E6POS: X 705.1693, Y 26.1098, Z -90.0150, A 0, B 90, C 0, E1 0, E2 0, E3 0, E4 0 } C_DIS
LIN{ E6POS: X 705.1698, Y 26.1746, Z -90.0150, A 0, B 90, C 0, E1 0, E2 0, E3 0, E4 0 } C_DIS
LIN{ E6POS: X 705.1921, Y 26.9713, Z -90.0150, A 0, B 90, C 0, E1 0, E2 0, E3 0, E4 0 } C_DIS
LIN{ E6POS: X 705.2363, Y 27.9703, Z -90.0150, A 0, B 90, C 0, E1 0, E2 0, E3 0, E4 0 } C_DIS
LIN{ E6POS: X 705.2513, Y 28.3073, Z -90.0150, A 0, B 90, C 0, E1 0, E2 0, E3 0, E4 0 } C_DIS
LIN{ E6POS: X 705.2912, Y 29.3065, Z -90.0150, A 0, B 90, C 0, E1 0, E2 0, E3 0, E4 0 } C_DIS
LIN{ E6POS: X 705.3050, Y 29.6503, Z -90.0150, A 0, B 90, C 0, E1 0, E2 0, E3 0, E4 0 } C_DIS
LIN{ E6POS: X 705.3050, Y 30.6503, Z -90.0150, A 0, B 90, C 0, E1 0, E2 0, E3 0, E4 0 } C_DIS
LIN{ E6POS: X 705.3050, Y 30.8868, Z -90.0150, A 0, B 90, C 0, E1 0, E2 0, E3 0, E4 0 } C_DIS
LIN{ E6POS: X 705.3230, Y 31.8850, Z -90.0150, A 0, B 90, C 0, E1 0, E2 0, E3 0, E4 0 } C_DIS
LIN{ E6POS: X 705.3214, Y 32.5969, Z -90.0150, A 0, B 90, C 0, E1 0, E2 0, E3 0, E4 0 } C_DIS
LIN{ E6POS: X 705.3365, Y 33.5968, Z -90.0150, A 0, B 90, C 0, E1 0, E2 0, E3 0, E4 0 } C_DIS
LIN{ E6POS: X 705.3389, Y 33.7597, Z -90.0150, A 0, B 90, C 0, E1 0, E2 0, E3 0, E4 0 } C_DIS
LIN{ E6POS: X 705.3373, Y 34.4716, Z -90.0150, A 0, B 90, C 0, E1 0, E2 0, E3 0, E4 0 } C_DIS
LIN{ E6POS: X 705.3524, Y 35.4715, Z -90.0150, A 0, B 90, C 0, E1 0, E2 0, E3 0, E4 0 } C_DIS
LIN{ E6POS: X 705.3548, Y 35.6344, Z -90.0150, A 0, B 90, C 0, E1 0, E2 0, E3 0, E4 0 } C_DIS
LIN{ E6POS: X 705.3558, Y 36.6344, Z -90.0150, A 0, B 90, C 0, E1 0, E2 0, E3 0, E4 0 } C_DIS
LIN{ E6POS: X 705.3560, Y 36.8173, Z -90.0150, A 0, B 90, C 0, E1 0, E2 0, E3 0, E4 0 } C_DIS
LIN{ E6POS: X 705.3752, Y 37.8152, Z -90.0150, A 0, B 90, C 0, E1 0, E2 0, E3 0, E4 0 } C_DIS
LIN{ E6POS: X 705.4163, Y 38.8144, Z -90.0150, A 0, B 90, C 0, E1 0, E2 0, E3 0, E4 0 } C_DIS
LIN{ E6POS: X 705.4233, Y 38.9843, Z -90.0150, A 0, B 90, C 0, E1 0, E2 0, E3 0, E4 0 } C_DIS
LIN{ E6POS: X 705.4769, Y 39.9829, Z -90.0150, A 0, B 90, C 0, E1 0, E2 0, E3 0, E4 0 } C_DIS
LIN{ E6POS: X 705.4854, Y 40.1418, Z -90.0150, A 0, B 90, C 0, E1 0, E2 0, E3 0, E4 0 } C_DIS
LIN{ E6POS: X 705.5019, Y 41.1417, Z -90.0150, A 0, B 90, C 0, E1 0, E2 0, E3 0, E4 0 } C_DIS
LIN{ E6POS: X 705.5047, Y 41.3097, Z -90.0150, A 0, B 90, C 0, E1 0, E2 0, E3 0, E4 0 } C_DIS
LIN{ E6POS: X 705.5437, Y 42.2908, Z -90.0150, A 0, B 90, C 0, E1 0, E2 0, E3 0, E4 0 } C_DIS
LIN{ E6POS: X 705.5578, Y 43.0142, Z -90.0150, A 0, B 90, C 0, E1 0, E2 0, E3 0, E4 0 } C_DIS
LIN{ E6POS: X 705.5938, Y 44.0135, Z -90.0150, A 0, B 90, C 0, E1 0, E2 0, E3 0, E4 0 } C_DIS
LIN{ E6POS: X 705.6001, Y 44.1885, Z -90.0150, A 0, B 90, C 0, E1 0, E2 0, E3 0, E4 0 } C_DIS
LIN{ E6POS: X 705.6143, Y 44.9609, Z -90.0150, A 0, B 90, C 0, E1 0, E2 0, E3 0, E4 0 } C_DIS
LIN{ E6POS: X 705.6489, Y 45.9603, Z -90.0150, A 0, B 90, C 0, E1 0, E2 0, E3 0, E4 0 } C_DIS
LIN{ E6POS: X 705.6572, Y 46.2009, Z -90.0150, A 0, B 90, C 0, E1 0, E2 0, E3 0, E4 0 } C_DIS
LIN{ E6POS: X 705.6697, Y 46.9309, Z -90.0150, A 0, B 90, C 0, E1 0, E2 0, E3 0, E4 0 } C_DIS
LIN{ E6POS: X 705.7045, Y 47.9303, Z -90.0150, A 0, B 90, C 0, E1 0, E2 0, E3 0, E4 0 } C_DIS
LIN{ E6POS: X 705.7107, Y 48.1075, Z -90.0150, A 0, B 90, C 0, E1 0, E2 0, E3 0, E4 0 } C_DIS
LIN{ E6POS: X 705.7483, Y 49.0924, Z -90.0150, A 0, B 90, C 0, E1 0, E2 0, E3 0, E4 0 } C_DIS
LIN{ E6POS: X 705.7563, Y 49.6879, Z -90.0150, A 0, B 90, C 0, E1 0, E2 0, E3 0, E4 0 } C_DIS
LIN{ E6POS: X 705.7898, Y 50.5283, Z -90.0150, A 0, B 90, C 0, E1 0, E2 0, E3 0, E4 0 } C_DIS
LIN{ E6POS: X 705.7949, Y 51.0225, Z -90.0150, A 0, B 90, C 0, E1 0, E2 0, E3 0, E4 0 } C_DIS
LIN{ E6POS: X 705.8274, Y 51.7675, Z -90.0150, A 0, B 90, C 0, E1 0, E2 0, E3 0, E4 0 } C_DIS
LIN{ E6POS: X 705.8304, Y 52.1943, Z -90.0150, A 0, B 90, C 0, E1 0, E2 0, E3 0, E4 0 } C_DIS
LIN{ E6POS: X 705.8616, Y 52.8944, Z -90.0150, A 0, B 90, C 0, E1 0, E2 0, E3 0, E4 0 } C_DIS
LIN{ E6POS: X 705.8634, Y 53.2878, Z -90.0150, A 0, B 90, C 0, E1 0, E2 0, E3 0, E4 0 } C_DIS
LIN{ E6POS: X 706.2705, Y 53.1869, Z -90.0150, A 0, B 90, C 0, E1 0, E2 0, E3 0, E4 0 } C_DIS
LIN{ E6POS: X 706.9402, Y 53.0296, Z -90.0150, A 0, B 90, C 0, E1 0, E2 0, E3 0, E4 0 } C_DIS
LIN{ E6POS: X 707.9108, Y 52.7889, Z -90.0150, A 0, B 90, C 0, E1 0, E2 0, E3 0, E4 0 } C_DIS
LIN{ E6POS: X 708.1614, Y 52.7267, Z -90.0150, A 0, B 90, C 0, E1 0, E2 0, E3 0, E4 0 } C_DIS
LIN{ E6POS: X 709.1299, Y 52.4777, Z -90.0150, A 0, B 90, C 0, E1 0, E2 0, E3 0, E4 0 } C_DIS
LIN{ E6POS: X 710.0984, Y 52.2286, Z -90.0150, A 0, B 90, C 0, E1 0, E2 0, E3 0, E4 0 } C_DIS
LIN{ E6POS: X 710.1653, Y 52.2114, Z -90.0150, A 0, B 90, C 0, E1 0, E2 0, E3 0, E4 0 } C_DIS
LIN{ E6POS: X 711.1360, Y 51.9708, Z -90.0150, A 0, B 90, C 0, E1 0, E2 0, E3 0, E4 0 } C_DIS
LIN{ E6POS: X 712.1066, Y 51.7302, Z -90.0150, A 0, B 90, C 0, E1 0, E2 0, E3 0, E4 0 } C_DIS
LIN{ E6POS: X 712.6078, Y 51.6059, Z -90.0150, A 0, B 90, C 0, E1 0, E2 0, E3 0, E4 0 } C_DIS
LIN{ E6POS: X 713.5756, Y 51.3543, Z -90.0150, A 0, B 90, C 0, E1 0, E2 0, E3 0, E4 0 } C_DIS
LIN{ E6POS: X 714.5435, Y 51.1027, Z -90.0150, A 0, B 90, C 0, E1 0, E2 0, E3 0, E4 0 } C_DIS
LIN{ E6POS: X 715.5113, Y 50.8511, Z -90.0150, A 0, B 90, C 0, E1 0, E2 0, E3 0, E4 0 } C_DIS
LIN{ E6POS: X 716.4791, Y 50.5995, Z -90.0150, A 0, B 90, C 0, E1 0, E2 0, E3 0, E4 0 } C_DIS
LIN{ E6POS: X 716.6136, Y 50.5645, Z -90.0150, A 0, B 90, C 0, E1 0, E2 0, E3 0, E4 0 } C_DIS
LIN{ E6POS: X 717.5842, Y 50.3239, Z -90.0150, A 0, B 90, C 0, E1 0, E2 0, E3 0, E4 0 } C_DIS
LIN{ E6POS: X 718.5548, Y 50.0832, Z -90.0150, A 0, B 90, C 0, E1 0, E2 0, E3 0, E4 0 } C_DIS
LIN{ E6POS: X 719.5254, Y 49.8426, Z -90.0150, A 0, B 90, C 0, E1 0, E2 0, E3 0, E4 0 } C_DIS
LIN{ E6POS: X 720.4960, Y 49.6019, Z -90.0150, A 0, B 90, C 0, E1 0, E2 0, E3 0, E4 0 } C_DIS
LIN{ E6POS: X 720.6843, Y 49.5553, Z -90.0150, A 0, B 90, C 0, E1 0, E2 0, E3 0, E4 0 } C_DIS
LIN{ E6POS: X 721.6519, Y 49.3027, Z -90.0150, A 0, B 90, C 0, E1 0, E2 0, E3 0, E4 0 } C_DIS
LIN{ E6POS: X 722.6194, Y 49.0500, Z -90.0150, A 0, B 90, C 0, E1 0, E2 0, E3 0, E4 0 } C_DIS
LIN{ E6POS: X 723.5870, Y 48.7974, Z -90.0150, A 0, B 90, C 0, E1 0, E2 0, E3 0, E4 0 } C_DIS
LIN{ E6POS: X 724.5546, Y 48.5448, Z -90.0150, A 0, B 90, C 0, E1 0, E2 0, E3 0, E4 0 } C_DIS
LIN{ E6POS: X 725.5222, Y 48.2922, Z -90.0150, A 0, B 90, C 0, E1 0, E2 0, E3 0, E4 0 } C_DIS
LIN{ E6POS: X 726.4897, Y 48.0396, Z -90.0150, A 0, B 90, C 0, E1 0, E2 0, E3 0, E4 0 } C_DIS
LIN{ E6POS: X 727.3605, Y 47.8123, Z -90.0150, A 0, B 90, C 0, E1 0, E2 0, E3 0, E4 0 } C_DIS
LIN{ E6POS: X 728.3333, Y 47.5809, Z -90.0150, A 0, B 90, C 0, E1 0, E2 0, E3 0, E4 0 } C_DIS
LIN{ E6POS: X 729.3062, Y 47.3496, Z -90.0150, A 0, B 90, C 0, E1 0, E2 0, E3 0, E4 0 } C_DIS
LIN{ E6POS: X 730.2791, Y 47.1183, Z -90.0150, A 0, B 90, C 0, E1 0, E2 0, E3 0, E4 0 } C_DIS
LIN{ E6POS: X 731.2520, Y 46.8869, Z -90.0150, A 0, B 90, C 0, E1 0, E2 0, E3 0, E4 0 } C_DIS
LIN{ E6POS: X 732.2248, Y 46.6556, Z -90.0150, A 0, B 90, C 0, E1 0, E2 0, E3 0, E4 0 } C_DIS
LIN{ E6POS: X 732.3814, Y 46.6184, Z -90.0150, A 0, B 90, C 0, E1 0, E2 0, E3 0, E4 0 } C_DIS
LIN{ E6POS: X 733.3515, Y 46.3758, Z -90.0150, A 0, B 90, C 0, E1 0, E2 0, E3 0, E4 0 } C_DIS
LIN{ E6POS: X 734.3217, Y 46.1333, Z -90.0150, A 0, B 90, C 0, E1 0, E2 0, E3 0, E4 0 } C_DIS
LIN{ E6POS: X 735.2918, Y 45.8907, Z -90.0150, A 0, B 90, C 0, E1 0, E2 0, E3 0, E4 0 } C_DIS
LIN{ E6POS: X 736.2619, Y 45.6482, Z -90.0150, A 0, B 90, C 0, E1 0, E2 0, E3 0, E4 0 } C_DIS
LIN{ E6POS: X 737.2321, Y 45.4057, Z -90.0150, A 0, B 90, C 0, E1 0, E2 0, E3 0, E4 0 } C_DIS
LIN{ E6POS: X 738.2022, Y 45.1631, Z -90.0150, A 0, B 90, C 0, E1 0, E2 0, E3 0, E4 0 } C_DIS
LIN{ E6POS: X 739.1724, Y 44.9206, Z -90.0150, A 0, B 90, C 0, E1 0, E2 0, E3 0, E4 0 } C_DIS
LIN{ E6POS: X 740.1425, Y 44.6780, Z -90.0150, A 0, B 90, C 0, E1 0, E2 0, E3 0, E4 0 } C_DIS
LIN{ E6POS: X 740.6336, Y 44.5552, Z -90.0150, A 0, B 90, C 0, E1 0, E2 0, E3 0, E4 0 } C_DIS
LIN{ E6POS: X 741.6105, Y 44.3415, Z -90.0150, A 0, B 90, C 0, E1 0, E2 0, E3 0, E4 0 } C_DIS
LIN{ E6POS: X 742.5874, Y 44.1277, Z -90.0150, A 0, B 90, C 0, E1 0, E2 0, E3 0, E4 0 } C_DIS
LIN{ E6POS: X 743.5643, Y 43.9139, Z -90.0150, A 0, B 90, C 0, E1 0, E2 0, E3 0, E4 0 } C_DIS
LIN{ E6POS: X 744.5412, Y 43.7001, Z -90.0150, A 0, B 90, C 0, E1 0, E2 0, E3 0, E4 0 } C_DIS
LIN{ E6POS: X 745.5180, Y 43.4864, Z -90.0150, A 0, B 90, C 0, E1 0, E2 0, E3 0, E4 0 } C_DIS
LIN{ E6POS: X 745.9265, Y 43.3970, Z -90.0150, A 0, B 90, C 0, E1 0, E2 0, E3 0, E4 0 } C_DIS
LIN{ E6POS: X 746.9012, Y 43.1736, Z -90.0150, A 0, B 90, C 0, E1 0, E2 0, E3 0, E4 0 } C_DIS
LIN{ E6POS: X 747.8760, Y 42.9503, Z -90.0150, A 0, B 90, C 0, E1 0, E2 0, E3 0, E4 0 } C_DIS
LIN{ E6POS: X 748.8507, Y 42.7269, Z -90.0150, A 0, B 90, C 0, E1 0, E2 0, E3 0, E4 0 } C_DIS
LIN{ E6POS: X 749.8255, Y 42.5036, Z -90.0150, A 0, B 90, C 0, E1 0, E2 0, E3 0, E4 0 } C_DIS
LIN{ E6POS: X 750.8002, Y 42.2802, Z -90.0150, A 0, B 90, C 0, E1 0, E2 0, E3 0, E4 0 } C_DIS
LIN{ E6POS: X 751.7749, Y 42.0569, Z -90.0150, A 0, B 90, C 0, E1 0, E2 0, E3 0, E4 0 } C_DIS
LIN{ E6POS: X 752.7497, Y 41.8335, Z -90.0150, A 0, B 90, C 0, E1 0, E2 0, E3 0, E4 0 } C_DIS
LIN{ E6POS: X 753.7244, Y 41.6102, Z -90.0150, A 0, B 90, C 0, E1 0, E2 0, E3 0, E4 0 } C_DIS
LIN{ E6POS: X 754.6624, Y 41.3952, Z -90.0150, A 0, B 90, C 0, E1 0, E2 0, E3 0, E4 0 } C_DIS
LIN{ E6POS: X 755.6457, Y 41.2135, Z -90.0150, A 0, B 90, C 0, E1 0, E2 0, E3 0, E4 0 } C_DIS
LIN{ E6POS: X 756.6291, Y 41.0317, Z -90.0150, A 0, B 90, C 0, E1 0, E2 0, E3 0, E4 0 } C_DIS
LIN{ E6POS: X 757.6124, Y 40.8499, Z -90.0150, A 0, B 90, C 0, E1 0, E2 0, E3 0, E4 0 } C_DIS
LIN{ E6POS: X 758.5957, Y 40.6682, Z -90.0150, A 0, B 90, C 0, E1 0, E2 0, E3 0, E4 0 } C_DIS
LIN{ E6POS: X 759.5485, Y 40.4920, Z -90.0150, A 0, B 90, C 0, E1 0, E2 0, E3 0, E4 0 } C_DIS
LIN{ E6POS: X 760.5306, Y 40.3036, Z -90.0150, A 0, B 90, C 0, E1 0, E2 0, E3 0, E4 0 } C_DIS
LIN{ E6POS: X 761.5127, Y 40.1152, Z -90.0150, A 0, B 90, C 0, E1 0, E2 0, E3 0, E4 0 } C_DIS
LIN{ E6POS: X 762.4948, Y 39.9268, Z -90.0150, A 0, B 90, C 0, E1 0, E2 0, E3 0, E4 0 } C_DIS
LIN{ E6POS: X 763.4768, Y 39.7383, Z -90.0150, A 0, B 90, C 0, E1 0, E2 0, E3 0, E4 0 } C_DIS
LIN{ E6POS: X 764.4589, Y 39.5499, Z -90.0150, A 0, B 90, C 0, E1 0, E2 0, E3 0, E4 0 } C_DIS
LIN{ E6POS: X 765.4410, Y 39.3615, Z -90.0150, A 0, B 90, C 0, E1 0, E2 0, E3 0, E4 0 } C_DIS
LIN{ E6POS: X 766.4231, Y 39.1730, Z -90.0150, A 0, B 90, C 0, E1 0, E2 0, E3 0, E4 0 } C_DIS
LIN{ E6POS: X 767.4052, Y 38.9846, Z -90.0150, A 0, B 90, C 0, E1 0, E2 0, E3 0, E4 0 } C_DIS
LIN{ E6POS: X 767.6736, Y 38.9331, Z -90.0150, A 0, B 90, C 0, E1 0, E2 0, E3 0, E4 0 } C_DIS
LIN{ E6POS: X 768.6673, Y 38.8210, Z -90.0150, A 0, B 90, C 0, E1 0, E2 0, E3 0, E4 0 } C_DIS
LIN{ E6POS: X 769.6610, Y 38.7090, Z -90.0150, A 0, B 90, C 0, E1 0, E2 0, E3 0, E4 0 } C_DIS
LIN{ E6POS: X 770.6547, Y 38.5969, Z -90.0150, A 0, B 90, C 0, E1 0, E2 0, E3 0, E4 0 } C_DIS
LIN{ E6POS: X 771.4756, Y 38.5043, Z -90.0150, A 0, B 90, C 0, E1 0, E2 0, E3 0, E4 0 } C_DIS
LIN{ E6POS: X 772.4691, Y 38.3906, Z -90.0150, A 0, B 90, C 0, E1 0, E2 0, E3 0, E4 0 } C_DIS
LIN{ E6POS: X 773.4626, Y 38.2770, Z -90.0150, A 0, B 90, C 0, E1 0, E2 0, E3 0, E4 0 } C_DIS
LIN{ E6POS: X 774.4562, Y 38.1634, Z -90.0150, A 0, B 90, C 0, E1 0, E2 0, E3 0, E4 0 } C_DIS
LIN{ E6POS: X 775.4497, Y 38.0497, Z -90.0150, A 0, B 90, C 0, E1 0, E2 0, E3 0, E4 0 } C_DIS
LIN{ E6POS: X 776.4432, Y 37.9361, Z -90.0150, A 0, B 90, C 0, E1 0, E2 0, E3 0, E4 0 } C_DIS
LIN{ E6POS: X 777.4367, Y 37.8224, Z -90.0150, A 0, B 90, C 0, E1 0, E2 0, E3 0, E4 0 } C_DIS
LIN{ E6POS: X 777.8975, Y 37.7697, Z -90.0150, A 0, B 90, C 0, E1 0, E2 0, E3 0, E4 0 } C_DIS
LIN{ E6POS: X 778.8972, Y 37.7452, Z -90.0150, A 0, B 90, C 0, E1 0, E2 0, E3 0, E4 0 } C_DIS
LIN{ E6POS: X 779.8969, Y 37.7207, Z -90.0150, A 0, B 90, C 0, E1 0, E2 0, E3 0, E4 0 } C_DIS
LIN{ E6POS: X 780.8859, Y 37.6964, Z -90.0150, A 0, B 90, C 0, E1 0, E2 0, E3 0, E4 0 } C_DIS
LIN{ E6POS: X 781.8856, Y 37.6739, Z -90.0150, A 0, B 90, C 0, E1 0, E2 0, E3 0, E4 0 } C_DIS
LIN{ E6POS: X 782.8854, Y 37.6514, Z -90.0150, A 0, B 90, C 0, E1 0, E2 0, E3 0, E4 0 } C_DIS
LIN{ E6POS: X 783.8851, Y 37.6288, Z -90.0150, A 0, B 90, C 0, E1 0, E2 0, E3 0, E4 0 } C_DIS
LIN{ E6POS: X 784.8849, Y 37.6063, Z -90.0150, A 0, B 90, C 0, E1 0, E2 0, E3 0, E4 0 } C_DIS
LIN{ E6POS: X 785.8846, Y 37.5837, Z -90.0150, A 0, B 90, C 0, E1 0, E2 0, E3 0, E4 0 } C_DIS
LIN{ E6POS: X 786.0297, Y 37.5805, Z -90.0150, A 0, B 90, C 0, E1 0, E2 0, E3 0, E4 0 } C_DIS
LIN{ E6POS: X 787.0275, Y 37.6474, Z -90.0150, A 0, B 90, C 0, E1 0, E2 0, E3 0, E4 0 } C_DIS
LIN{ E6POS: X 788.0253, Y 37.7142, Z -90.0150, A 0, B 90, C 0, E1 0, E2 0, E3 0, E4 0 } C_DIS
LIN{ E6POS: X 788.4759, Y 37.7445, Z -90.0150, A 0, B 90, C 0, E1 0, E2 0, E3 0, E4 0 } C_DIS
LIN{ E6POS: X 789.4735, Y 37.8133, Z -90.0150, A 0, B 90, C 0, E1 0, E2 0, E3 0, E4 0 } C_DIS
LIN{ E6POS: X 790.4711, Y 37.8822, Z -90.0150, A 0, B 90, C 0, E1 0, E2 0, E3 0, E4 0 } C_DIS
LIN{ E6POS: X 791.4687, Y 37.9511, Z -90.0150, A 0, B 90, C 0, E1 0, E2 0, E3 0, E4 0 } C_DIS
LIN{ E6POS: X 792.4663, Y 38.0200, Z -90.0150, A 0, B 90, C 0, E1 0, E2 0, E3 0, E4 0 } C_DIS
LIN{ E6POS: X 792.7685, Y 38.0409, Z -90.0150, A 0, B 90, C 0, E1 0, E2 0, E3 0, E4 0 } C_DIS
LIN{ E6POS: X 793.7601, Y 38.1698, Z -90.0150, A 0, B 90, C 0, E1 0, E2 0, E3 0, E4 0 } C_DIS
LIN{ E6POS: X 794.7518, Y 38.2986, Z -90.0150, A 0, B 90, C 0, E1 0, E2 0, E3 0, E4 0 } C_DIS
LIN{ E6POS: X 794.9433, Y 38.3235, Z -90.0150, A 0, B 90, C 0, E1 0, E2 0, E3 0, E4 0 } C_DIS
LIN{ E6POS: X 795.9350, Y 38.4524, Z -90.0150, A 0, B 90, C 0, E1 0, E2 0, E3 0, E4 0 } C_DIS
LIN{ E6POS: X 796.9266, Y 38.5813, Z -90.0150, A 0, B 90, C 0, E1 0, E2 0, E3 0, E4 0 } C_DIS
LIN{ E6POS: X 797.9183, Y 38.7102, Z -90.0150, A 0, B 90, C 0, E1 0, E2 0, E3 0, E4 0 } C_DIS
LIN{ E6POS: X 798.8097, Y 38.8260, Z -88.0150, A 0, B 90, C 0, E1 0, E2 0, E3 0, E4 0 } C_DIS
LIN{ E6POS: X 798.7068, Y 37.8313, Z -88.0150, A 0, B 90, C 0, E1 0, E2 0, E3 0, E4 0 } C_DIS
LIN{ E6POS: X 798.6040, Y 36.8366, Z -88.0150, A 0, B 90, C 0, E1 0, E2 0, E3 0, E4 0 } C_DIS
LIN{ E6POS: X 798.5012, Y 35.8419, Z -88.0150, A 0, B 90, C 0, E1 0, E2 0, E3 0, E4 0 } C_DIS
LIN{ E6POS: X 798.3983, Y 34.8472, Z -88.0150, A 0, B 90, C 0, E1 0, E2 0, E3 0, E4 0 } C_DIS
LIN{ E6POS: X 798.2955, Y 33.8525, Z -88.0150, A 0, B 90, C 0, E1 0, E2 0, E3 0, E4 0 } C_DIS
LIN{ E6POS: X 798.1927, Y 32.8578, Z -88.0150, A 0, B 90, C 0, E1 0, E2 0, E3 0, E4 0 } C_DIS
LIN{ E6POS: X 798.0898, Y 31.8631, Z -88.0150, A 0, B 90, C 0, E1 0, E2 0, E3 0, E4 0 } C_DIS
LIN{ E6POS: X 798.0673, Y 31.6448, Z -88.0150, A 0, B 90, C 0, E1 0, E2 0, E3 0, E4 0 } C_DIS
LIN{ E6POS: X 797.9644, Y 30.6501, Z -88.0150, A 0, B 90, C 0, E1 0, E2 0, E3 0, E4 0 } C_DIS
LIN{ E6POS: X 797.8616, Y 29.6554, Z -88.0150, A 0, B 90, C 0, E1 0, E2 0, E3 0, E4 0 } C_DIS
LIN{ E6POS: X 797.7588, Y 28.6607, Z -88.0150, A 0, B 90, C 0, E1 0, E2 0, E3 0, E4 0 } C_DIS
LIN{ E6POS: X 797.6559, Y 27.6660, Z -88.0150, A 0, B 90, C 0, E1 0, E2 0, E3 0, E4 0 } C_DIS
LIN{ E6POS: X 797.5531, Y 26.6713, Z -88.0150, A 0, B 90, C 0, E1 0, E2 0, E3 0, E4 0 } C_DIS
LIN{ E6POS: X 797.4503, Y 25.6766, Z -88.0150, A 0, B 90, C 0, E1 0, E2 0, E3 0, E4 0 } C_DIS
LIN{ E6POS: X 797.3474, Y 24.6819, Z -88.0150, A 0, B 90, C 0, E1 0, E2 0, E3 0, E4 0 } C_DIS
LIN{ E6POS: X 797.2446, Y 23.6872, Z -88.0150, A 0, B 90, C 0, E1 0, E2 0, E3 0, E4 0 } C_DIS
LIN{ E6POS: X 797.1418, Y 22.6925, Z -88.0150, A 0, B 90, C 0, E1 0, E2 0, E3 0, E4 0 } C_DIS
LIN{ E6POS: X 797.1224, Y 22.5051, Z -88.0150, A 0, B 90, C 0, E1 0, E2 0, E3 0, E4 0 } C_DIS
LIN{ E6POS: X 797.0002, Y 21.5126, Z -88.0150, A 0, B 90, C 0, E1 0, E2 0, E3 0, E4 0 } C_DIS
LIN{ E6POS: X 796.8780, Y 20.5201, Z -88.0150, A 0, B 90, C 0, E1 0, E2 0, E3 0, E4 0 } C_DIS
LIN{ E6POS: X 796.7559, Y 19.5276, Z -88.0150, A 0, B 90, C 0, E1 0, E2 0, E3 0, E4 0 } C_DIS
LIN{ E6POS: X 796.6337, Y 18.5351, Z -88.0150, A 0, B 90, C 0, E1 0, E2 0, E3 0, E4 0 } C_DIS
LIN{ E6POS: X 796.5115, Y 17.5426, Z -88.0150, A 0, B 90, C 0, E1 0, E2 0, E3 0, E4 0 } C_DIS
LIN{ E6POS: X 796.3893, Y 16.5500, Z -88.0150, A 0, B 90, C 0, E1 0, E2 0, E3 0, E4 0 } C_DIS
LIN{ E6POS: X 796.3013, Y 15.8348, Z -88.0150, A 0, B 90, C 0, E1 0, E2 0, E3 0, E4 0 } C_DIS
LIN{ E6POS: X 796.1791, Y 14.8423, Z -88.0150, A 0, B 90, C 0, E1 0, E2 0, E3 0, E4 0 } C_DIS
LIN{ E6POS: X 796.0569, Y 13.8497, Z -88.0150, A 0, B 90, C 0, E1 0, E2 0, E3 0, E4 0 } C_DIS
LIN{ E6POS: X 795.9348, Y 12.8572, Z -88.0150, A 0, B 90, C 0, E1 0, E2 0, E3 0, E4 0 } C_DIS
LIN{ E6POS: X 795.8126, Y 11.8647, Z -88.0150, A 0, B 90, C 0, E1 0, E2 0, E3 0, E4 0 } C_DIS
LIN{ E6POS: X 795.6904, Y 10.8722, Z -88.0150, A 0, B 90, C 0, E1 0, E2 0, E3 0, E4 0 } C_DIS
LIN{ E6POS: X 795.5682, Y 9.8797, Z -88.0150, A 0, B 90, C 0, E1 0, E2 0, E3 0, E4 0 } C_DIS
LIN{ E6POS: X 795.4460, Y 8.8872, Z -88.0150, A 0, B 90, C 0, E1 0, E2 0, E3 0, E4 0 } C_DIS
LIN{ E6POS: X 795.3239, Y 7.8947, Z -88.0150, A 0, B 90, C 0, E1 0, E2 0, E3 0, E4 0 } C_DIS
LIN{ E6POS: X 795.2562, Y 7.3452, Z -88.0150, A 0, B 90, C 0, E1 0, E2 0, E3 0, E4 0 } C_DIS
LIN{ E6POS: X 795.0854, Y 6.3599, Z -88.0150, A 0, B 90, C 0, E1 0, E2 0, E3 0, E4 0 } C_DIS
LIN{ E6POS: X 794.9146, Y 5.3746, Z -88.0150, A 0, B 90, C 0, E1 0, E2 0, E3 0, E4 0 } C_DIS
LIN{ E6POS: X 794.7438, Y 4.3893, Z -88.0150, A 0, B 90, C 0, E1 0, E2 0, E3 0, E4 0 } C_DIS
LIN{ E6POS: X 794.5730, Y 3.4040, Z -88.0150, A 0, B 90, C 0, E1 0, E2 0, E3 0, E4 0 } C_DIS
LIN{ E6POS: X 794.4021, Y 2.4187, Z -88.0150, A 0, B 90, C 0, E1 0, E2 0, E3 0, E4 0 } C_DIS
LIN{ E6POS: X 794.2771, Y 1.6977, Z -88.0150, A 0, B 90, C 0, E1 0, E2 0, E3 0, E4 0 } C_DIS
LIN{ E6POS: X 794.1063, Y 0.7124, Z -88.0150, A 0, B 90, C 0, E1 0, E2 0, E3 0, E4 0 } C_DIS
LIN{ E6POS: X 793.9355, Y -0.2729, Z -88.0150, A 0, B 90, C 0, E1 0, E2 0, E3 0, E4 0 } C_DIS
LIN{ E6POS: X 793.7647, Y -1.2582, Z -88.0150, A 0, B 90, C 0, E1 0, E2 0, E3 0, E4 0 } C_DIS
LIN{ E6POS: X 793.5939, Y -2.2435, Z -88.0150, A 0, B 90, C 0, E1 0, E2 0, E3 0, E4 0 } C_DIS
LIN{ E6POS: X 793.4231, Y -3.2288, Z -88.0150, A 0, B 90, C 0, E1 0, E2 0, E3 0, E4 0 } C_DIS
LIN{ E6POS: X 793.2522, Y -4.2141, Z -88.0150, A 0, B 90, C 0, E1 0, E2 0, E3 0, E4 0 } C_DIS
LIN{ E6POS: X 793.0814, Y -5.1994, Z -88.0150, A 0, B 90, C 0, E1 0, E2 0, E3 0, E4 0 } C_DIS
LIN{ E6POS: X 793.0310, Y -5.4900, Z -88.0150, A 0, B 90, C 0, E1 0, E2 0, E3 0, E4 0 } C_DIS
LIN{ E6POS: X 792.7476, Y -6.4490, Z -88.0150, A 0, B 90, C 0, E1 0, E2 0, E3 0, E4 0 } C_DIS
LIN{ E6POS: X 792.4642, Y -7.4080, Z -88.0150, A 0, B 90, C 0, E1 0, E2 0, E3 0, E4 0 } C_DIS
LIN{ E6POS: X 792.1808, Y -8.3670, Z -88.0150, A 0, B 90, C 0, E1 0, E2 0, E3 0, E4 0 } C_DIS
LIN{ E6POS: X 791.8974, Y -9.3260, Z -88.0150, A 0, B 90, C 0, E1 0, E2 0, E3 0, E4 0 } C_DIS
LIN{ E6POS: X 791.8154, Y -9.6035, Z -88.0150, A 0, B 90, C 0, E1 0, E2 0, E3 0, E4 0 } C_DIS
LIN{ E6POS: X 791.5319, Y -10.5625, Z -88.0150, A 0, B 90, C 0, E1 0, E2 0, E3 0, E4 0 } C_DIS
LIN{ E6POS: X 791.2485, Y -11.5215, Z -88.0150, A 0, B 90, C 0, E1 0, E2 0, E3 0, E4 0 } C_DIS
LIN{ E6POS: X 790.9651, Y -12.4805, Z -88.0150, A 0, B 90, C 0, E1 0, E2 0, E3 0, E4 0 } C_DIS
LIN{ E6POS: X 790.6817, Y -13.4395, Z -88.0150, A 0, B 90, C 0, E1 0, E2 0, E3 0, E4 0 } C_DIS
LIN{ E6POS: X 790.3983, Y -14.3985, Z -88.0150, A 0, B 90, C 0, E1 0, E2 0, E3 0, E4 0 } C_DIS
LIN{ E6POS: X 790.2681, Y -14.8387, Z -88.0150, A 0, B 90, C 0, E1 0, E2 0, E3 0, E4 0 } C_DIS
LIN{ E6POS: X 789.6733, Y -15.6426, Z -88.0150, A 0, B 90, C 0, E1 0, E2 0, E3 0, E4 0 } C_DIS
LIN{ E6POS: X 789.0784, Y -16.4464, Z -88.0150, A 0, B 90, C 0, E1 0, E2 0, E3 0, E4 0 } C_DIS
LIN{ E6POS: X 788.7371, Y -16.9076, Z -88.0150, A 0, B 90, C 0, E1 0, E2 0, E3 0, E4 0 } C_DIS
LIN{ E6POS: X 788.1422, Y -17.7115, Z -88.0150, A 0, B 90, C 0, E1 0, E2 0, E3 0, E4 0 } C_DIS
LIN{ E6POS: X 787.5473, Y -18.5153, Z -88.0150, A 0, B 90, C 0, E1 0, E2 0, E3 0, E4 0 } C_DIS
LIN{ E6POS: X 786.9525, Y -19.3191, Z -88.0150, A 0, B 90, C 0, E1 0, E2 0, E3 0, E4 0 } C_DIS
LIN{ E6POS: X 786.7884, Y -19.5408, Z -88.0150, A 0, B 90, C 0, E1 0, E2 0, E3 0, E4 0 } C_DIS
LIN{ E6POS: X 785.8300, Y -19.8262, Z -88.0150, A 0, B 90, C 0, E1 0, E2 0, E3 0, E4 0 } C_DIS
LIN{ E6POS: X 784.8717, Y -20.1117, Z -88.0150, A 0, B 90, C 0, E1 0, E2 0, E3 0, E4 0 } C_DIS
LIN{ E6POS: X 784.8157, Y -20.1284, Z -88.0150, A 0, B 90, C 0, E1 0, E2 0, E3 0, E4 0 } C_DIS
LIN{ E6POS: X 783.8584, Y -20.4176, Z -88.0150, A 0, B 90, C 0, E1 0, E2 0, E3 0, E4 0 } C_DIS
LIN{ E6POS: X 782.9012, Y -20.7068, Z -88.0150, A 0, B 90, C 0, E1 0, E2 0, E3 0, E4 0 } C_DIS
LIN{ E6POS: X 782.3374, Y -20.8771, Z -88.0150, A 0, B 90, C 0, E1 0, E2 0, E3 0, E4 0 } C_DIS
LIN{ E6POS: X 781.3461, Y -20.7455, Z -88.0150, A 0, B 90, C 0, E1 0, E2 0, E3 0, E4 0 } C_DIS
LIN{ E6POS: X 780.3548, Y -20.6139, Z -88.0150, A 0, B 90, C 0, E1 0, E2 0, E3 0, E4 0 } C_DIS
LIN{ E6POS: X 779.3635, Y -20.4823, Z -88.0150, A 0, B 90, C 0, E1 0, E2 0, E3 0, E4 0 } C_DIS
LIN{ E6POS: X 779.2030, Y -20.4610, Z -88.0150, A 0, B 90, C 0, E1 0, E2 0, E3 0, E4 0 } C_DIS
LIN{ E6POS: X 778.2113, Y -20.3324, Z -88.0150, A 0, B 90, C 0, E1 0, E2 0, E3 0, E4 0 } C_DIS
LIN{ E6POS: X 777.2196, Y -20.2039, Z -88.0150, A 0, B 90, C 0, E1 0, E2 0, E3 0, E4 0 } C_DIS
LIN{ E6POS: X 776.6629, Y -20.1317, Z -88.0150, A 0, B 90, C 0, E1 0, E2 0, E3 0, E4 0 } C_DIS
LIN{ E6POS: X 775.6863, Y -19.9169, Z -88.0150, A 0, B 90, C 0, E1 0, E2 0, E3 0, E4 0 } C_DIS
LIN{ E6POS: X 774.7096, Y -19.7020, Z -88.0150, A 0, B 90, C 0, E1 0, E2 0, E3 0, E4 0 } C_DIS
LIN{ E6POS: X 773.7330, Y -19.4871, Z -88.0150, A 0, B 90, C 0, E1 0, E2 0, E3 0, E4 0 } C_DIS
LIN{ E6POS: X 772.7563, Y -19.2722, Z -88.0150, A 0, B 90, C 0, E1 0, E2 0, E3 0, E4 0 } C_DIS
LIN{ E6POS: X 772.7439, Y -19.2695, Z -88.0150, A 0, B 90, C 0, E1 0, E2 0, E3 0, E4 0 } C_DIS
LIN{ E6POS: X 771.7654, Y -19.0630, Z -88.0150, A 0, B 90, C 0, E1 0, E2 0, E3 0, E4 0 } C_DIS
LIN{ E6POS: X 770.7870, Y -18.8565, Z -88.0150, A 0, B 90, C 0, E1 0, E2 0, E3 0, E4 0 } C_DIS
LIN{ E6POS: X 769.8085, Y -18.6500, Z -88.0150, A 0, B 90, C 0, E1 0, E2 0, E3 0, E4 0 } C_DIS
LIN{ E6POS: X 769.5101, Y -18.5870, Z -88.0150, A 0, B 90, C 0, E1 0, E2 0, E3 0, E4 0 } C_DIS
LIN{ E6POS: X 768.5174, Y -18.4659, Z -88.0150, A 0, B 90, C 0, E1 0, E2 0, E3 0, E4 0 } C_DIS
LIN{ E6POS: X 767.5248, Y -18.3448, Z -88.0150, A 0, B 90, C 0, E1 0, E2 0, E3 0, E4 0 } C_DIS
LIN{ E6POS: X 766.5321, Y -18.2236, Z -88.0150, A 0, B 90, C 0, E1 0, E2 0, E3 0, E4 0 } C_DIS
LIN{ E6POS: X 765.5395, Y -18.1025, Z -88.0150, A 0, B 90, C 0, E1 0, E2 0, E3 0, E4 0 } C_DIS
LIN{ E6POS: X 764.6795, Y -17.9975, Z -88.0150, A 0, B 90, C 0, E1 0, E2 0, E3 0, E4 0 } C_DIS
LIN{ E6POS: X 763.6862, Y -17.8820, Z -88.0150, A 0, B 90, C 0, E1 0, E2 0, E3 0, E4 0 } C_DIS
LIN{ E6POS: X 762.6929, Y -17.7666, Z -88.0150, A 0, B 90, C 0, E1 0, E2 0, E3 0, E4 0 } C_DIS
LIN{ E6POS: X 761.6996, Y -17.6511, Z -88.0150, A 0, B 90, C 0, E1 0, E2 0, E3 0, E4 0 } C_DIS
LIN{ E6POS: X 760.7062, Y -17.5356, Z -88.0150, A 0, B 90, C 0, E1 0, E2 0, E3 0, E4 0 } C_DIS
LIN{ E6POS: X 760.6266, Y -17.5264, Z -88.0150, A 0, B 90, C 0, E1 0, E2 0, E3 0, E4 0 } C_DIS
LIN{ E6POS: X 759.6287, Y -17.4616, Z -88.0150, A 0, B 90, C 0, E1 0, E2 0, E3 0, E4 0 } C_DIS
LIN{ E6POS: X 758.6308, Y -17.3969, Z -88.0150, A 0, B 90, C 0, E1 0, E2 0, E3 0, E4 0 } C_DIS
LIN{ E6POS: X 757.6329, Y -17.3322, Z -88.0150, A 0, B 90, C 0, E1 0, E2 0, E3 0, E4 0 } C_DIS
LIN{ E6POS: X 756.6350, Y -17.2674, Z -88.0150, A 0, B 90, C 0, E1 0, E2 0, E3 0, E4 0 } C_DIS
LIN{ E6POS: X 755.6371, Y -17.2027, Z -88.0150, A 0, B 90, C 0, E1 0, E2 0, E3 0, E4 0 } C_DIS
LIN{ E6POS: X 755.4995, Y -17.1938, Z -88.0150, A 0, B 90, C 0, E1 0, E2 0, E3 0, E4 0 } C_DIS
LIN{ E6POS: X 754.5014, Y -17.1311, Z -88.0150, A 0, B 90, C 0, E1 0, E2 0, E3 0, E4 0 } C_DIS
LIN{ E6POS: X 753.5034, Y -17.0684, Z -88.0150, A 0, B 90, C 0, E1 0, E2 0, E3 0, E4 0 } C_DIS
LIN{ E6POS: X 752.5054, Y -17.0057, Z -88.0150, A 0, B 90, C 0, E1 0, E2 0, E3 0, E4 0 } C_DIS
LIN{ E6POS: X 751.5073, Y -16.9430, Z -88.0150, A 0, B 90, C 0, E1 0, E2 0, E3 0, E4 0 } C_DIS
LIN{ E6POS: X 751.1626, Y -16.9213, Z -88.0150, A 0, B 90, C 0, E1 0, E2 0, E3 0, E4 0 } C_DIS
LIN{ E6POS: X 750.1627, Y -16.9024, Z -88.0150, A 0, B 90, C 0, E1 0, E2 0, E3 0, E4 0 } C_DIS
LIN{ E6POS: X 749.1629, Y -16.8835, Z -88.0150, A 0, B 90, C 0, E1 0, E2 0, E3 0, E4 0 } C_DIS
LIN{ E6POS: X 748.1631, Y -16.8646, Z -88.0150, A 0, B 90, C 0, E1 0, E2 0, E3 0, E4 0 } C_DIS
LIN{ E6POS: X 747.1633, Y -16.8457, Z -88.0150, A 0, B 90, C 0, E1 0, E2 0, E3 0, E4 0 } C_DIS
LIN{ E6POS: X 746.3535, Y -16.8304, Z -88.0150, A 0, B 90, C 0, E1 0, E2 0, E3 0, E4 0 } C_DIS
LIN{ E6POS: X 745.3538, Y -16.8092, Z -88.0150, A 0, B 90, C 0, E1 0, E2 0, E3 0, E4 0 } C_DIS
LIN{ E6POS: X 744.3540, Y -16.7880, Z -88.0150, A 0, B 90, C 0, E1 0, E2 0, E3 0, E4 0 } C_DIS
LIN{ E6POS: X 743.3542, Y -16.7668, Z -88.0150, A 0, B 90, C 0, E1 0, E2 0, E3 0, E4 0 } C_DIS
LIN{ E6POS: X 742.3544, Y -16.7455, Z -88.0150, A 0, B 90, C 0, E1 0, E2 0, E3 0, E4 0 } C_DIS
LIN{ E6POS: X 742.2677, Y -16.7437, Z -88.0150, A 0, B 90, C 0, E1 0, E2 0, E3 0, E4 0 } C_DIS
LIN{ E6POS: X 741.2683, Y -16.7783, Z -88.0150, A 0, B 90, C 0, E1 0, E2 0, E3 0, E4 0 } C_DIS
LIN{ E6POS: X 740.2689, Y -16.8129, Z -88.0150, A 0, B 90, C 0, E1 0, E2 0, E3 0, E4 0 } C_DIS
LIN{ E6POS: X 739.2695, Y -16.8475, Z -88.0150, A 0, B 90, C 0, E1 0, E2 0, E3 0, E4 0 } C_DIS
LIN{ E6POS: X 738.3925, Y -16.8778, Z -88.0150, A 0, B 90, C 0, E1 0, E2 0, E3 0, E4 0 } C_DIS
LIN{ E6POS: X 737.3928, Y -16.9040, Z -88.0150, A 0, B 90, C 0, E1 0, E2 0, E3 0, E4 0 } C_DIS
LIN{ E6POS: X 736.3931, Y -16.9302, Z -88.0150, A 0, B 90, C 0, E1 0, E2 0, E3 0, E4 0 } C_DIS
LIN{ E6POS: X 735.3935, Y -16.9563, Z -88.0150, A 0, B 90, C 0, E1 0, E2 0, E3 0, E4 0 } C_DIS
LIN{ E6POS: X 735.0927, Y -16.9642, Z -88.0150, A 0, B 90, C 0, E1 0, E2 0, E3 0, E4 0 } C_DIS
LIN{ E6POS: X 734.1035, Y -17.1107, Z -88.0150, A 0, B 90, C 0, E1 0, E2 0, E3 0, E4 0 } C_DIS
LIN{ E6POS: X 733.1143, Y -17.2573, Z -88.0150, A 0, B 90, C 0, E1 0, E2 0, E3 0, E4 0 } C_DIS
LIN{ E6POS: X 732.7664, Y -17.3088, Z -88.0150, A 0, B 90, C 0, E1 0, E2 0, E3 0, E4 0 } C_DIS
LIN{ E6POS: X 731.7741, Y -17.4327, Z -88.0150, A 0, B 90, C 0, E1 0, E2 0, E3 0, E4 0 } C_DIS
LIN{ E6POS: X 730.7880, Y -17.5558, Z -88.0150, A 0, B 90, C 0, E1 0, E2 0, E3 0, E4 0 } C_DIS
LIN{ E6POS: X 730.0103, Y -18.1061, Z -88.0150, A 0, B 90, C 0, E1 0, E2 0, E3 0, E4 0 } C_DIS
LIN{ E6POS: X 729.3521, Y -18.5155, Z -88.0150, A 0, B 90, C 0, E1 0, E2 0, E3 0, E4 0 } C_DIS
LIN{ E6POS: X 730.0123, Y -19.0892, Z -88.0150, A 0, B 90, C 0, E1 0, E2 0, E3 0, E4 0 } C_DIS
LIN{ E6POS: X 730.7289, Y -19.7867, Z -88.0150, A 0, B 90, C 0, E1 0, E2 0, E3 0, E4 0 } C_DIS
LIN{ E6POS: X 730.7830, Y -19.8395, Z -88.0150, A 0, B 90, C 0, E1 0, E2 0, E3 0, E4 0 } C_DIS
LIN{ E6POS: X 731.7195, Y -20.1902, Z -88.0150, A 0, B 90, C 0, E1 0, E2 0, E3 0, E4 0 } C_DIS
LIN{ E6POS: X 732.6559, Y -20.5410, Z -88.0150, A 0, B 90, C 0, E1 0, E2 0, E3 0, E4 0 } C_DIS
LIN{ E6POS: X 732.7609, Y -20.5803, Z -88.0150, A 0, B 90, C 0, E1 0, E2 0, E3 0, E4 0 } C_DIS
LIN{ E6POS: X 733.6868, Y -20.9582, Z -88.0150, A 0, B 90, C 0, E1 0, E2 0, E3 0, E4 0 } C_DIS
LIN{ E6POS: X 734.6126, Y -21.3361, Z -88.0150, A 0, B 90, C 0, E1 0, E2 0, E3 0, E4 0 } C_DIS
LIN{ E6POS: X 735.0800, Y -21.5269, Z -88.0150, A 0, B 90, C 0, E1 0, E2 0, E3 0, E4 0 } C_DIS
LIN{ E6POS: X 736.0439, Y -21.7930, Z -88.0150, A 0, B 90, C 0, E1 0, E2 0, E3 0, E4 0 } C_DIS
LIN{ E6POS: X 737.0079, Y -22.0592, Z -88.0150, A 0, B 90, C 0, E1 0, E2 0, E3 0, E4 0 } C_DIS
LIN{ E6POS: X 737.9718, Y -22.3253, Z -88.0150, A 0, B 90, C 0, E1 0, E2 0, E3 0, E4 0 } C_DIS
LIN{ E6POS: X 738.3739, Y -22.4363, Z -88.0150, A 0, B 90, C 0, E1 0, E2 0, E3 0, E4 0 } C_DIS
LIN{ E6POS: X 739.3333, Y -22.7187, Z -88.0150, A 0, B 90, C 0, E1 0, E2 0, E3 0, E4 0 } C_DIS
LIN{ E6POS: X 740.2926, Y -23.0010, Z -88.0150, A 0, B 90, C 0, E1 0, E2 0, E3 0, E4 0 } C_DIS
LIN{ E6POS: X 741.2519, Y -23.2834, Z -88.0150, A 0, B 90, C 0, E1 0, E2 0, E3 0, E4 0 } C_DIS
LIN{ E6POS: X 742.2112, Y -23.5657, Z -88.0150, A 0, B 90, C 0, E1 0, E2 0, E3 0, E4 0 } C_DIS
LIN{ E6POS: X 742.2405, Y -23.5743, Z -88.0150, A 0, B 90, C 0, E1 0, E2 0, E3 0, E4 0 } C_DIS
LIN{ E6POS: X 743.2153, Y -23.7973, Z -88.0150, A 0, B 90, C 0, E1 0, E2 0, E3 0, E4 0 } C_DIS
LIN{ E6POS: X 744.1902, Y -24.0203, Z -88.0150, A 0, B 90, C 0, E1 0, E2 0, E3 0, E4 0 } C_DIS
LIN{ E6POS: X 745.1650, Y -24.2432, Z -88.0150, A 0, B 90, C 0, E1 0, E2 0, E3 0, E4 0 } C_DIS
LIN{ E6POS: X 746.1398, Y -24.4662, Z -88.0150, A 0, B 90, C 0, E1 0, E2 0, E3 0, E4 0 } C_DIS
LIN{ E6POS: X 746.3185, Y -24.5071, Z -88.0150, A 0, B 90, C 0, E1 0, E2 0, E3 0, E4 0 } C_DIS
LIN{ E6POS: X 747.2908, Y -24.7405, Z -88.0150, A 0, B 90, C 0, E1 0, E2 0, E3 0, E4 0 } C_DIS
LIN{ E6POS: X 748.2632, Y -24.9739, Z -88.0150, A 0, B 90, C 0, E1 0, E2 0, E3 0, E4 0 } C_DIS
LIN{ E6POS: X 749.2356, Y -25.2073, Z -88.0150, A 0, B 90, C 0, E1 0, E2 0, E3 0, E4 0 } C_DIS
LIN{ E6POS: X 750.2079, Y -25.4408, Z -88.0150, A 0, B 90, C 0, E1 0, E2 0, E3 0, E4 0 } C_DIS
LIN{ E6POS: X 751.1197, Y -25.6596, Z -88.0150, A 0, B 90, C 0, E1 0, E2 0, E3 0, E4 0 } C_DIS
LIN{ E6POS: X 752.1027, Y -25.8434, Z -88.0150, A 0, B 90, C 0, E1 0, E2 0, E3 0, E4 0 } C_DIS
LIN{ E6POS: X 753.0856, Y -26.0271, Z -88.0150, A 0, B 90, C 0, E1 0, E2 0, E3 0, E4 0 } C_DIS
LIN{ E6POS: X 754.0686, Y -26.2109, Z -88.0150, A 0, B 90, C 0, E1 0, E2 0, E3 0, E4 0 } C_DIS
LIN{ E6POS: X 755.0516, Y -26.3946, Z -88.0150, A 0, B 90, C 0, E1 0, E2 0, E3 0, E4 0 } C_DIS
LIN{ E6POS: X 755.4487, Y -26.4688, Z -88.0150, A 0, B 90, C 0, E1 0, E2 0, E3 0, E4 0 } C_DIS
LIN{ E6POS: X 756.4304, Y -26.6588, Z -88.0150, A 0, B 90, C 0, E1 0, E2 0, E3 0, E4 0 } C_DIS
LIN{ E6POS: X 757.4122, Y -26.8488, Z -88.0150, A 0, B 90, C 0, E1 0, E2 0, E3 0, E4 0 } C_DIS
LIN{ E6POS: X 758.3940, Y -27.0388, Z -88.0150, A 0, B 90, C 0, E1 0, E2 0, E3 0, E4 0 } C_DIS
LIN{ E6POS: X 759.3758, Y -27.2288, Z -88.0150, A 0, B 90, C 0, E1 0, E2 0, E3 0, E4 0 } C_DIS
LIN{ E6POS: X 760.3576, Y -27.4188, Z -88.0150, A 0, B 90, C 0, E1 0, E2 0, E3 0, E4 0 } C_DIS
LIN{ E6POS: X 760.5710, Y -27.4601, Z -88.0150, A 0, B 90, C 0, E1 0, E2 0, E3 0, E4 0 } C_DIS
LIN{ E6POS: X 761.5622, Y -27.5924, Z -88.0150, A 0, B 90, C 0, E1 0, E2 0, E3 0, E4 0 } C_DIS
LIN{ E6POS: X 762.5534, Y -27.7248, Z -88.0150, A 0, B 90, C 0, E1 0, E2 0, E3 0, E4 0 } C_DIS
LIN{ E6POS: X 763.5446, Y -27.8571, Z -88.0150, A 0, B 90, C 0, E1 0, E2 0, E3 0, E4 0 } C_DIS
LIN{ E6POS: X 764.5358, Y -27.9894, Z -88.0150, A 0, B 90, C 0, E1 0, E2 0, E3 0, E4 0 } C_DIS
LIN{ E6POS: X 764.6188, Y -28.0005, Z -88.0150, A 0, B 90, C 0, E1 0, E2 0, E3 0, E4 0 } C_DIS
LIN{ E6POS: X 765.6098, Y -28.1345, Z -88.0150, A 0, B 90, C 0, E1 0, E2 0, E3 0, E4 0 } C_DIS
LIN{ E6POS: X 766.6008, Y -28.2686, Z -88.0150, A 0, B 90, C 0, E1 0, E2 0, E3 0, E4 0 } C_DIS
LIN{ E6POS: X 767.5918, Y -28.4026, Z -88.0150, A 0, B 90, C 0, E1 0, E2 0, E3 0, E4 0 } C_DIS
LIN{ E6POS: X 768.5828, Y -28.5366, Z -88.0150, A 0, B 90, C 0, E1 0, E2 0, E3 0, E4 0 } C_DIS
LIN{ E6POS: X 769.4478, Y -28.6536, Z -88.0150, A 0, B 90, C 0, E1 0, E2 0, E3 0, E4 0 } C_DIS
LIN{ E6POS: X 770.4471, Y -28.6923, Z -88.0150, A 0, B 90, C 0, E1 0, E2 0, E3 0, E4 0 } C_DIS
LIN{ E6POS: X 771.4463, Y -28.7309, Z -88.0150, A 0, B 90, C 0, E1 0, E2 0, E3 0, E4 0 } C_DIS
LIN{ E6POS: X 772.4456, Y -28.7696, Z -88.0150, A 0, B 90, C 0, E1 0, E2 0, E3 0, E4 0 } C_DIS
LIN{ E6POS: X 772.6824, Y -28.7787, Z -88.0150, A 0, B 90, C 0, E1 0, E2 0, E3 0, E4 0 } C_DIS
LIN{ E6POS: X 773.6818, Y -28.8143, Z -88.0150, A 0, B 90, C 0, E1 0, E2 0, E3 0, E4 0 } C_DIS
LIN{ E6POS: X 774.6812, Y -28.8498, Z -88.0150, A 0, B 90, C 0, E1 0, E2 0, E3 0, E4 0 } C_DIS
LIN{ E6POS: X 775.6805, Y -28.8853, Z -88.0150, A 0, B 90, C 0, E1 0, E2 0, E3 0, E4 0 } C_DIS
LIN{ E6POS: X 776.6060, Y -28.9182, Z -88.0150, A 0, B 90, C 0, E1 0, E2 0, E3 0, E4 0 } C_DIS
LIN{ E6POS: X 777.5895, Y -29.0989, Z -88.0150, A 0, B 90, C 0, E1 0, E2 0, E3 0, E4 0 } C_DIS
LIN{ E6POS: X 778.5730, Y -29.2797, Z -88.0150, A 0, B 90, C 0, E1 0, E2 0, E3 0, E4 0 } C_DIS
LIN{ E6POS: X 778.9718, Y -29.3530, Z -88.0150, A 0, B 90, C 0, E1 0, E2 0, E3 0, E4 0 } C_DIS
LIN{ E6POS: X 779.9549, Y -29.5358, Z -88.0150, A 0, B 90, C 0, E1 0, E2 0, E3 0, E4 0 } C_DIS
LIN{ E6POS: X 780.9381, Y -29.7187, Z -88.0150, A 0, B 90, C 0, E1 0, E2 0, E3 0, E4 0 } C_DIS
LIN{ E6POS: X 781.8855, Y -29.8950, Z -88.0150, A 0, B 90, C 0, E1 0, E2 0, E3 0, E4 0 } C_DIS
LIN{ E6POS: X 782.5862, Y -30.6085, Z -88.0150, A 0, B 90, C 0, E1 0, E2 0, E3 0, E4 0 } C_DIS
LIN{ E6POS: X 783.2868, Y -31.3220, Z -88.0150, A 0, B 90, C 0, E1 0, E2 0, E3 0, E4 0 } C_DIS
LIN{ E6POS: X 783.3263, Y -31.3622, Z -88.0150, A 0, B 90, C 0, E1 0, E2 0, E3 0, E4 0 } C_DIS
LIN{ E6POS: X 784.0212, Y -32.0813, Z -88.0150, A 0, B 90, C 0, E1 0, E2 0, E3 0, E4 0 } C_DIS
LIN{ E6POS: X 784.7162, Y -32.8004, Z -88.0150, A 0, B 90, C 0, E1 0, E2 0, E3 0, E4 0 } C_DIS
LIN{ E6POS: X 785.1281, Y -33.2266, Z -88.0150, A 0, B 90, C 0, E1 0, E2 0, E3 0, E4 0 } C_DIS
LIN{ E6POS: X 785.2695, Y -34.2166, Z -88.0150, A 0, B 90, C 0, E1 0, E2 0, E3 0, E4 0 } C_DIS
LIN{ E6POS: X 785.4109, Y -35.2065, Z -88.0150, A 0, B 90, C 0, E1 0, E2 0, E3 0, E4 0 } C_DIS
LIN{ E6POS: X 785.5523, Y -36.1965, Z -88.0150, A 0, B 90, C 0, E1 0, E2 0, E3 0, E4 0 } C_DIS
LIN{ E6POS: X 785.5886, Y -36.4505, Z -88.0150, A 0, B 90, C 0, E1 0, E2 0, E3 0, E4 0 } C_DIS
LIN{ E6POS: X 785.7300, Y -37.4404, Z -88.0150, A 0, B 90, C 0, E1 0, E2 0, E3 0, E4 0 } C_DIS
LIN{ E6POS: X 785.8714, Y -38.4304, Z -88.0150, A 0, B 90, C 0, E1 0, E2 0, E3 0, E4 0 } C_DIS
LIN{ E6POS: X 786.0128, Y -39.4203, Z -88.0150, A 0, B 90, C 0, E1 0, E2 0, E3 0, E4 0 } C_DIS
LIN{ E6POS: X 786.1542, Y -40.4103, Z -88.0150, A 0, B 90, C 0, E1 0, E2 0, E3 0, E4 0 } C_DIS
LIN{ E6POS: X 786.1747, Y -40.5536, Z -88.0150, A 0, B 90, C 0, E1 0, E2 0, E3 0, E4 0 } C_DIS
LIN{ E6POS: X 786.0743, Y -41.5485, Z -88.0150, A 0, B 90, C 0, E1 0, E2 0, E3 0, E4 0 } C_DIS
LIN{ E6POS: X 785.9740, Y -42.5435, Z -88.0150, A 0, B 90, C 0, E1 0, E2 0, E3 0, E4 0 } C_DIS
LIN{ E6POS: X 785.8737, Y -43.5384, Z -88.0150, A 0, B 90, C 0, E1 0, E2 0, E3 0, E4 0 } C_DIS
LIN{ E6POS: X 785.7734, Y -44.5334, Z -88.0150, A 0, B 90, C 0, E1 0, E2 0, E3 0, E4 0 } C_DIS
LIN{ E6POS: X 785.6731, Y -45.5283, Z -88.0150, A 0, B 90, C 0, E1 0, E2 0, E3 0, E4 0 } C_DIS
LIN{ E6POS: X 785.5995, Y -46.2581, Z -88.0150, A 0, B 90, C 0, E1 0, E2 0, E3 0, E4 0 } C_DIS
LIN{ E6POS: X 785.4992, Y -47.2531, Z -88.0150, A 0, B 90, C 0, E1 0, E2 0, E3 0, E4 0 } C_DIS
LIN{ E6POS: X 785.3989, Y -48.2480, Z -88.0150, A 0, B 90, C 0, E1 0, E2 0, E3 0, E4 0 } C_DIS
LIN{ E6POS: X 785.2986, Y -49.2430, Z -88.0150, A 0, B 90, C 0, E1 0, E2 0, E3 0, E4 0 } C_DIS
LIN{ E6POS: X 785.1983, Y -50.2379, Z -88.0150, A 0, B 90, C 0, E1 0, E2 0, E3 0, E4 0 } C_DIS
LIN{ E6POS: X 785.0979, Y -51.2329, Z -88.0150, A 0, B 90, C 0, E1 0, E2 0, E3 0, E4 0 } C_DIS
LIN{ E6POS: X 784.9976, Y -52.2278, Z -88.0150, A 0, B 90, C 0, E1 0, E2 0, E3 0, E4 0 } C_DIS
LIN{ E6POS: X 784.8973, Y -53.2228, Z -88.0150, A 0, B 90, C 0, E1 0, E2 0, E3 0, E4 0 } C_DIS
LIN{ E6POS: X 784.8675, Y -53.5185, Z -88.0150, A 0, B 90, C 0, E1 0, E2 0, E3 0, E4 0 } C_DIS
LIN{ E6POS: X 784.6915, Y -54.5029, Z -88.0150, A 0, B 90, C 0, E1 0, E2 0, E3 0, E4 0 } C_DIS
LIN{ E6POS: X 784.5156, Y -55.4873, Z -88.0150, A 0, B 90, C 0, E1 0, E2 0, E3 0, E4 0 } C_DIS
LIN{ E6POS: X 784.3396, Y -56.4717, Z -88.0150, A 0, B 90, C 0, E1 0, E2 0, E3 0, E4 0 } C_DIS
LIN{ E6POS: X 784.1637, Y -57.4560, Z -88.0150, A 0, B 90, C 0, E1 0, E2 0, E3 0, E4 0 } C_DIS
LIN{ E6POS: X 783.9877, Y -58.4404, Z -88.0150, A 0, B 90, C 0, E1 0, E2 0, E3 0, E4 0 } C_DIS
LIN{ E6POS: X 783.8118, Y -59.4248, Z -88.0150, A 0, B 90, C 0, E1 0, E2 0, E3 0, E4 0 } C_DIS
LIN{ E6POS: X 783.6358, Y -60.4092, Z -88.0150, A 0, B 90, C 0, E1 0, E2 0, E3 0, E4 0 } C_DIS
LIN{ E6POS: X 783.5153, Y -61.0835, Z -88.0150, A 0, B 90, C 0, E1 0, E2 0, E3 0, E4 0 } C_DIS
LIN{ E6POS: X 783.3394, Y -62.0679, Z -88.0150, A 0, B 90, C 0, E1 0, E2 0, E3 0, E4 0 } C_DIS
LIN{ E6POS: X 783.1634, Y -63.0523, Z -88.0150, A 0, B 90, C 0, E1 0, E2 0, E3 0, E4 0 } C_DIS
LIN{ E6POS: X 782.9875, Y -64.0367, Z -88.0150, A 0, B 90, C 0, E1 0, E2 0, E3 0, E4 0 } C_DIS
LIN{ E6POS: X 782.8115, Y -65.0211, Z -88.0150, A 0, B 90, C 0, E1 0, E2 0, E3 0, E4 0 } C_DIS
LIN{ E6POS: X 782.6356, Y -66.0055, Z -88.0150, A 0, B 90, C 0, E1 0, E2 0, E3 0, E4 0 } C_DIS
LIN{ E6POS: X 782.4596, Y -66.9899, Z -88.0150, A 0, B 90, C 0, E1 0, E2 0, E3 0, E4 0 } C_DIS
LIN{ E6POS: X 782.2836, Y -67.9743, Z -88.0150, A 0, B 90, C 0, E1 0, E2 0, E3 0, E4 0 } C_DIS
LIN{ E6POS: X 782.1077, Y -68.9587, Z -88.0150, A 0, B 90, C 0, E1 0, E2 0, E3 0, E4 0 } C_DIS
LIN{ E6POS: X 781.9317, Y -69.9431, Z -88.0150, A 0, B 90, C 0, E1 0, E2 0, E3 0, E4 0 } C_DIS
LIN{ E6POS: X 781.7943, Y -70.7119, Z -88.0150, A 0, B 90, C 0, E1 0, E2 0, E3 0, E4 0 } C_DIS
LIN{ E6POS: X 781.5865, Y -71.6900, Z -88.0150, A 0, B 90, C 0, E1 0, E2 0, E3 0, E4 0 } C_DIS
LIN{ E6POS: X 781.3787, Y -72.6682, Z -88.0150, A 0, B 90, C 0, E1 0, E2 0, E3 0, E4 0 } C_DIS
LIN{ E6POS: X 781.1709, Y -73.6464, Z -88.0150, A 0, B 90, C 0, E1 0, E2 0, E3 0, E4 0 } C_DIS
LIN{ E6POS: X 780.9631, Y -74.6245, Z -88.0150, A 0, B 90, C 0, E1 0, E2 0, E3 0, E4 0 } C_DIS
LIN{ E6POS: X 780.7553, Y -75.6027, Z -88.0150, A 0, B 90, C 0, E1 0, E2 0, E3 0, E4 0 } C_DIS
LIN{ E6POS: X 780.5475, Y -76.5809, Z -88.0150, A 0, B 90, C 0, E1 0, E2 0, E3 0, E4 0 } C_DIS
LIN{ E6POS: X 780.3397, Y -77.5590, Z -88.0150, A 0, B 90, C 0, E1 0, E2 0, E3 0, E4 0 } C_DIS
LIN{ E6POS: X 780.1319, Y -78.5372, Z -88.0150, A 0, B 90, C 0, E1 0, E2 0, E3 0, E4 0 } C_DIS
LIN{ E6POS: X 779.9241, Y -79.5154, Z -88.0150, A 0, B 90, C 0, E1 0, E2 0, E3 0, E4 0 } C_DIS
LIN{ E6POS: X 779.9237, Y -79.5173, Z -88.0150, A 0, B 90, C 0, E1 0, E2 0, E3 0, E4 0 } C_DIS
LIN{ E6POS: X 779.7159, Y -80.4955, Z -88.0150, A 0, B 90, C 0, E1 0, E2 0, E3 0, E4 0 } C_DIS
LIN{ E6POS: X 779.5081, Y -81.4737, Z -88.0150, A 0, B 90, C 0, E1 0, E2 0, E3 0, E4 0 } C_DIS
LIN{ E6POS: X 779.3003, Y -82.4518, Z -88.0150, A 0, B 90, C 0, E1 0, E2 0, E3 0, E4 0 } C_DIS
LIN{ E6POS: X 779.0925, Y -83.4300, Z -88.0150, A 0, B 90, C 0, E1 0, E2 0, E3 0, E4 0 } C_DIS
LIN{ E6POS: X 778.8847, Y -84.4082, Z -88.0150, A 0, B 90, C 0, E1 0, E2 0, E3 0, E4 0 } C_DIS
LIN{ E6POS: X 778.6769, Y -85.3863, Z -88.0150, A 0, B 90, C 0, E1 0, E2 0, E3 0, E4 0 } C_DIS
LIN{ E6POS: X 778.4691, Y -86.3645, Z -88.0150, A 0, B 90, C 0, E1 0, E2 0, E3 0, E4 0 } C_DIS
LIN{ E6POS: X 778.2613, Y -87.3427, Z -88.0150, A 0, B 90, C 0, E1 0, E2 0, E3 0, E4 0 } C_DIS
LIN{ E6POS: X 778.0535, Y -88.3209, Z -88.0150, A 0, B 90, C 0, E1 0, E2 0, E3 0, E4 0 } C_DIS
LIN{ E6POS: X 777.8457, Y -89.2990, Z -88.0150, A 0, B 90, C 0, E1 0, E2 0, E3 0, E4 0 } C_DIS
LIN{ E6POS: X 777.6379, Y -90.2772, Z -88.0150, A 0, B 90, C 0, E1 0, E2 0, E3 0, E4 0 } C_DIS
LIN{ E6POS: X 777.5429, Y -90.7243, Z -88.0150, A 0, B 90, C 0, E1 0, E2 0, E3 0, E4 0 } C_DIS
LIN{ E6POS: X 777.3226, Y -91.6997, Z -88.0150, A 0, B 90, C 0, E1 0, E2 0, E3 0, E4 0 } C_DIS
LIN{ E6POS: X 777.1022, Y -92.6751, Z -88.0150, A 0, B 90, C 0, E1 0, E2 0, E3 0, E4 0 } C_DIS
LIN{ E6POS: X 776.8819, Y -93.6506, Z -88.0150, A 0, B 90, C 0, E1 0, E2 0, E3 0, E4 0 } C_DIS
LIN{ E6POS: X 776.6615, Y -94.6260, Z -88.0150, A 0, B 90, C 0, E1 0, E2 0, E3 0, E4 0 } C_DIS
LIN{ E6POS: X 776.4412, Y -95.6014, Z -88.0150, A 0, B 90, C 0, E1 0, E2 0, E3 0, E4 0 } C_DIS
LIN{ E6POS: X 776.2208, Y -96.5768, Z -88.0150, A 0, B 90, C 0, E1 0, E2 0, E3 0, E4 0 } C_DIS
LIN{ E6POS: X 776.0005, Y -97.5522, Z -88.0150, A 0, B 90, C 0, E1 0, E2 0, E3 0, E4 0 } C_DIS
LIN{ E6POS: X 775.7802, Y -98.5277, Z -88.0150, A 0, B 90, C 0, E1 0, E2 0, E3 0, E4 0 } C_DIS
LIN{ E6POS: X 775.5598, Y -99.5031, Z -88.0150, A 0, B 90, C 0, E1 0, E2 0, E3 0, E4 0 } C_DIS
LIN{ E6POS: X 775.4137, Y -100.1499, Z -88.0150, A 0, B 90, C 0, E1 0, E2 0, E3 0, E4 0 } C_DIS
LIN{ E6POS: X 775.1933, Y -101.1254, Z -88.0150, A 0, B 90, C 0, E1 0, E2 0, E3 0, E4 0 } C_DIS
LIN{ E6POS: X 774.9730, Y -102.1008, Z -88.0150, A 0, B 90, C 0, E1 0, E2 0, E3 0, E4 0 } C_DIS
LIN{ E6POS: X 774.7527, Y -103.0762, Z -88.0150, A 0, B 90, C 0, E1 0, E2 0, E3 0, E4 0 } C_DIS
LIN{ E6POS: X 774.5323, Y -104.0516, Z -88.0150, A 0, B 90, C 0, E1 0, E2 0, E3 0, E4 0 } C_DIS
LIN{ E6POS: X 774.3120, Y -105.0270, Z -88.0150, A 0, B 90, C 0, E1 0, E2 0, E3 0, E4 0 } C_DIS
LIN{ E6POS: X 774.0916, Y -106.0025, Z -88.0150, A 0, B 90, C 0, E1 0, E2 0, E3 0, E4 0 } C_DIS
LIN{ E6POS: X 773.8713, Y -106.9779, Z -88.0150, A 0, B 90, C 0, E1 0, E2 0, E3 0, E4 0 } C_DIS
LIN{ E6POS: X 773.6509, Y -107.9533, Z -88.0150, A 0, B 90, C 0, E1 0, E2 0, E3 0, E4 0 } C_DIS
LIN{ E6POS: X 773.4306, Y -108.9287, Z -88.0150, A 0, B 90, C 0, E1 0, E2 0, E3 0, E4 0 } C_DIS
LIN{ E6POS: X 773.2102, Y -109.9041, Z -88.0150, A 0, B 90, C 0, E1 0, E2 0, E3 0, E4 0 } C_DIS
LIN{ E6POS: X 772.9899, Y -110.8796, Z -88.0150, A 0, B 90, C 0, E1 0, E2 0, E3 0, E4 0 } C_DIS
LIN{ E6POS: X 772.7695, Y -111.8550, Z -88.0150, A 0, B 90, C 0, E1 0, E2 0, E3 0, E4 0 } C_DIS
LIN{ E6POS: X 772.7038, Y -112.1462, Z -88.0150, A 0, B 90, C 0, E1 0, E2 0, E3 0, E4 0 } C_DIS
LIN{ E6POS: X 772.0412, Y -111.3972, Z -88.0150, A 0, B 90, C 0, E1 0, E2 0, E3 0, E4 0 } C_DIS
LIN{ E6POS: X 771.5280, Y -110.8169, Z -88.0150, A 0, B 90, C 0, E1 0, E2 0, E3 0, E4 0 } C_DIS
LIN{ E6POS: X 770.8655, Y -110.0678, Z -88.0150, A 0, B 90, C 0, E1 0, E2 0, E3 0, E4 0 } C_DIS
LIN{ E6POS: X 770.2029, Y -109.3188, Z -88.0150, A 0, B 90, C 0, E1 0, E2 0, E3 0, E4 0 } C_DIS
LIN{ E6POS: X 770.0315, Y -109.1250, Z -88.0150, A 0, B 90, C 0, E1 0, E2 0, E3 0, E4 0 } C_DIS
LIN{ E6POS: X 769.2888, Y -108.4553, Z -88.0150, A 0, B 90, C 0, E1 0, E2 0, E3 0, E4 0 } C_DIS
LIN{ E6POS: X 768.5461, Y -107.7857, Z -88.0150, A 0, B 90, C 0, E1 0, E2 0, E3 0, E4 0 } C_DIS
LIN{ E6POS: X 768.4806, Y -107.7266, Z -88.0150, A 0, B 90, C 0, E1 0, E2 0, E3 0, E4 0 } C_DIS
LIN{ E6POS: X 767.7388, Y -107.0560, Z -88.0150, A 0, B 90, C 0, E1 0, E2 0, E3 0, E4 0 } C_DIS
LIN{ E6POS: X 766.9969, Y -106.3854, Z -88.0150, A 0, B 90, C 0, E1 0, E2 0, E3 0, E4 0 } C_DIS
